// TIA Portal V15.1 export
// export: Created 2024-06-21T08:41:07.2186582Z, ExportSetting WithDefaults, DisplayName Totally Integrated Automation Portal, DisplayVersion V15.1 Update 5, DisplayName TIA Portal Openness, DisplayVersion V15.1 Update 5, DisplayName SINAMICS Startdrive Advanced, DisplayVersion V15.1, DisplayName G130, G150, S120, S150, SINAMICS MV, S210, DisplayVersion V15.1, DisplayName G110M, G120, G120C, G120D, G120P, DisplayVersion V15.1, DisplayName STEP 7 Professional, DisplayVersion V15.1 Update 5, DisplayName STEP 7 Safety, DisplayVersion V15.1, DisplayName WinCC Professional, DisplayVersion V15.1 Update 5, DisplayName SIMATIC Visualization Architect, DisplayVersion V15.1
FUNCTION_BLOCK "LGBHandHeldHBA"   // FB6712, FBD
TITLE = LGBHandHeldHBA
{ S7_Optimized_Access := 'FALSE' }
AUTHOR : VCG
FAMILY : OPanel
VERSION : 1.0
// stored: AutoNumber false, IsIECCheckEnabled false, SetENOAutomatically False, UDAEnableTagReadback false
   VAR_INPUT
      I_HMINbrHandHeld { ExternalAccessible := 'False'; ExternalVisible := 'False'; ExternalWritable := 'False'} : Int;   // HMI number on the function block ModeSelectorHW
      I_ActiveHMI { ExternalAccessible := 'False'; ExternalVisible := 'False'; ExternalWritable := 'False'} : Int;   // Active HMI in the ModeSelectorHW
      I_Connected { ExternalAccessible := 'False'; ExternalVisible := 'False'; ExternalWritable := 'False'} : Bool;   // HandHeld is connected
      I_DeathmansSwitch { ExternalAccessible := 'False'; ExternalVisible := 'False'; ExternalWritable := 'False'} : Bool;   // Deathmans switch
      I_PBSet { ExternalAccessible := 'False'; ExternalVisible := 'False'; ExternalWritable := 'False'} : Bool;   // Push button for manual movememt -> set
      I_PBReset { ExternalAccessible := 'False'; ExternalVisible := 'False'; ExternalWritable := 'False'} : Bool;   // Push button for manual movememt -> reset
      I_PBAlarmReset { ExternalAccessible := 'False'; ExternalVisible := 'False'; ExternalWritable := 'False'} : Bool;   // Push button Alarm reset / Alarm reset pushbutton is activated
      "I_PBSpeed+" { ExternalAccessible := 'False'; ExternalVisible := 'False'; ExternalWritable := 'False'} : Bool;   // Puls for Speed+
      "I_PBSpeed-" { ExternalAccessible := 'False'; ExternalVisible := 'False'; ExternalWritable := 'False'} : Bool;   // Puls for Speed-
      I_PBSelectDevice1 { ExternalAccessible := 'False'; ExternalVisible := 'False'; ExternalWritable := 'False'} : Bool;   // Push button for select Device 1
      I_PBSelectDevice2 { ExternalAccessible := 'False'; ExternalVisible := 'False'; ExternalWritable := 'False'} : Bool;   // Push button for select Device 2
      I_PBSelectDevice3 { ExternalAccessible := 'False'; ExternalVisible := 'False'; ExternalWritable := 'False'} : Bool;   // Push button for select Device 3
      I_PBSelectDevice4 { ExternalAccessible := 'False'; ExternalVisible := 'False'; ExternalWritable := 'False'} : Bool;   // Push button for select Device 4
      I_PBSelectDevice5 { ExternalAccessible := 'False'; ExternalVisible := 'False'; ExternalWritable := 'False'} : Bool;   // Push button for select Device 5
      I_PBSelectDevice6 { ExternalAccessible := 'False'; ExternalVisible := 'False'; ExternalWritable := 'False'} : Bool;   // Push button for select Device 6
      I_PBSelectDevice7 { ExternalAccessible := 'False'; ExternalVisible := 'False'; ExternalWritable := 'False'} : Bool;   // Push button for select Device7
      I_PBSelectDevice8 { ExternalAccessible := 'False'; ExternalVisible := 'False'; ExternalWritable := 'False'} : Bool;   // Push button for select Device 8
      I_PBSelectDevice9 { ExternalAccessible := 'False'; ExternalVisible := 'False'; ExternalWritable := 'False'} : Bool;   // Push button for select Device 9
      I_ActiveDevice1 { ExternalAccessible := 'False'; ExternalVisible := 'False'; ExternalWritable := 'False'} : Bool;   // Device 1 is active
      I_ActiveDevice2 { ExternalAccessible := 'False'; ExternalVisible := 'False'; ExternalWritable := 'False'} : Bool;   // Device 2 is active
      I_ActiveDevice3 { ExternalAccessible := 'False'; ExternalVisible := 'False'; ExternalWritable := 'False'} : Bool;   // Device 3 is active
      I_ActiveDevice4 { ExternalAccessible := 'False'; ExternalVisible := 'False'; ExternalWritable := 'False'} : Bool;   // Device 4 is active
      I_ActiveDevice5 { ExternalAccessible := 'False'; ExternalVisible := 'False'; ExternalWritable := 'False'} : Bool;   // Device 5 is active
      I_ActiveDevice6 { ExternalAccessible := 'False'; ExternalVisible := 'False'; ExternalWritable := 'False'} : Bool;   // Device 6 is active
      I_ActiveDevice7 { ExternalAccessible := 'False'; ExternalVisible := 'False'; ExternalWritable := 'False'} : Bool;   // Device 7 is active
      I_ActiveDevice8 { ExternalAccessible := 'False'; ExternalVisible := 'False'; ExternalWritable := 'False'} : Bool;   // Device 8 is active
      I_ActiveDevice9 { ExternalAccessible := 'False'; ExternalVisible := 'False'; ExternalWritable := 'False'} : Bool;   // Device 9 is active
      I_LEDAlarmReset { ExternalAccessible := 'False'; ExternalVisible := 'False'; ExternalWritable := 'False'} : Bool;   // Led Indication Push button Alarm reset / Alarm reset pushbutton is activated
   END_VAR
   VAR_OUTPUT
      O_HandHeldConnected { ExternalAccessible := 'False'; ExternalVisible := 'False'; ExternalWritable := 'False'} : Bool;   // HandHeld is connected
      O_HandHeldSelected { ExternalAccessible := 'False'; ExternalVisible := 'False'; ExternalWritable := 'False'} : Bool;   // HandHeld is selected, is active HMI
      O_AlarmReset { ExternalAccessible := 'False'; ExternalVisible := 'False'; ExternalWritable := 'False'} : Bool;   // Push button Alarm reset / Alarm reset pushbutton is activated
      O_Speed { ExternalAccessible := 'False'; ExternalVisible := 'False'; ExternalWritable := 'False'} : Int;   // Speed
      "O_Speed+" { ExternalAccessible := 'False'; ExternalVisible := 'False'; ExternalWritable := 'False'} : Bool;   // Push button Speed+
      "O_Speed-" { ExternalAccessible := 'False'; ExternalVisible := 'False'; ExternalWritable := 'False'} : Bool;   // Push button Speed-
      O_HighSpeed { ExternalAccessible := 'False'; ExternalVisible := 'False'; ExternalWritable := 'False'} : Bool;   // High Speed Selected
      O_PBSetDevice1 { ExternalAccessible := 'False'; ExternalVisible := 'False'; ExternalWritable := 'False'} : Bool;   // Device 1 Push button Set
      O_PBResDevice1 { ExternalAccessible := 'False'; ExternalVisible := 'False'; ExternalWritable := 'False'} : Bool;   // Device 1 Push button Reset
      O_PBSetDevice2 { ExternalAccessible := 'False'; ExternalVisible := 'False'; ExternalWritable := 'False'} : Bool;   // Device 2 Push button Set
      O_PBResDevice2 { ExternalAccessible := 'False'; ExternalVisible := 'False'; ExternalWritable := 'False'} : Bool;   // Device 2 Push button Reset
      O_PBSetDevice3 { ExternalAccessible := 'False'; ExternalVisible := 'False'; ExternalWritable := 'False'} : Bool;   // Device 3 Push button Set
      O_PBResDevice3 { ExternalAccessible := 'False'; ExternalVisible := 'False'; ExternalWritable := 'False'} : Bool;   // Device 3 Push button Reset
      O_PBSetDevice4 { ExternalAccessible := 'False'; ExternalVisible := 'False'; ExternalWritable := 'False'} : Bool;   // Device 4 Push button Set
      O_PBResDevice4 { ExternalAccessible := 'False'; ExternalVisible := 'False'; ExternalWritable := 'False'} : Bool;   // Device 4 Push button Reset
      O_PBSetDevice5 { ExternalAccessible := 'False'; ExternalVisible := 'False'; ExternalWritable := 'False'} : Bool;   // Device 5 Push button Set
      O_PBResDevice5 { ExternalAccessible := 'False'; ExternalVisible := 'False'; ExternalWritable := 'False'} : Bool;   // Device 5 Push button Reset
      O_PBSetDevice6 { ExternalAccessible := 'False'; ExternalVisible := 'False'; ExternalWritable := 'False'} : Bool;   // Device 6 Push button Set
      O_PBResDevice6 { ExternalAccessible := 'False'; ExternalVisible := 'False'; ExternalWritable := 'False'} : Bool;   // Device 6 Push button Reset
      O_PBSetDevice7 { ExternalAccessible := 'False'; ExternalVisible := 'False'; ExternalWritable := 'False'} : Bool;   // Device 7 Push button Set
      O_PBResDevice7 { ExternalAccessible := 'False'; ExternalVisible := 'False'; ExternalWritable := 'False'} : Bool;   // Device 7 Push button Reset
      O_PBSetDevice8 { ExternalAccessible := 'False'; ExternalVisible := 'False'; ExternalWritable := 'False'} : Bool;   // Device 8 Push button Set
      O_PBResDevice8 { ExternalAccessible := 'False'; ExternalVisible := 'False'; ExternalWritable := 'False'} : Bool;   // Device 8 Push button Reset
      O_PBSetDevice9 { ExternalAccessible := 'False'; ExternalVisible := 'False'; ExternalWritable := 'False'} : Bool;   // Device 9 Push button Set
      O_PBResDevice9 { ExternalAccessible := 'False'; ExternalVisible := 'False'; ExternalWritable := 'False'} : Bool;   // Device 9 Push button Reset
      O_LEDSet { ExternalAccessible := 'False'; ExternalVisible := 'False'; ExternalWritable := 'False'} : Bool;   // Led Indication Push button set
      O_LEDReset { ExternalAccessible := 'False'; ExternalVisible := 'False'; ExternalWritable := 'False'} : Bool;   // Led Indication Push button reset
      O_LEDAlarmReset { ExternalAccessible := 'False'; ExternalVisible := 'False'; ExternalWritable := 'False'} : Bool;   // Led Indication Push button Alarm reset / Alarm reset pushbutton is activated
      "O_LEDSpeed+" { ExternalAccessible := 'False'; ExternalVisible := 'False'; ExternalWritable := 'False'} : Bool;   // Led Indication Puls Speed+
      "O_LEDSpeed-" { ExternalAccessible := 'False'; ExternalVisible := 'False'; ExternalWritable := 'False'} : Bool;   // Led Indication Puls Speed-
      O_LEDDevice1 { ExternalAccessible := 'False'; ExternalVisible := 'False'; ExternalWritable := 'False'} : Bool;   // Led Indication Push button Device 1
      O_LEDDevice2 { ExternalAccessible := 'False'; ExternalVisible := 'False'; ExternalWritable := 'False'} : Bool;   // Led Indication Push button Device 2
      O_LEDDevice3 { ExternalAccessible := 'False'; ExternalVisible := 'False'; ExternalWritable := 'False'} : Bool;   // Led Indication Push button Device 3
      O_LEDDevice4 { ExternalAccessible := 'False'; ExternalVisible := 'False'; ExternalWritable := 'False'} : Bool;   // Led Indication Push button Device 4
      O_LEDDevice5 { ExternalAccessible := 'False'; ExternalVisible := 'False'; ExternalWritable := 'False'} : Bool;   // Led Indication Push button Device 5
      O_LEDDevice6 { ExternalAccessible := 'False'; ExternalVisible := 'False'; ExternalWritable := 'False'} : Bool;   // Led Indication Push button Device 6
      O_LEDDevice7 { ExternalAccessible := 'False'; ExternalVisible := 'False'; ExternalWritable := 'False'} : Bool;   // Led Indication Push button Device 7
      O_LEDDevice8 { ExternalAccessible := 'False'; ExternalVisible := 'False'; ExternalWritable := 'False'} : Bool;   // Led Indication Push button Device 8
      O_LEDDevice9 { ExternalAccessible := 'False'; ExternalVisible := 'False'; ExternalWritable := 'False'} : Bool;   // Led Indication Push button Device 9
   END_VAR
   VAR_IN_OUT
      IO_Modes : "Modes";   // Modes IO
      C_Config : "HandHeldHBA-Config";   // Config
   END_VAR
   VAR DB_SPECIFIC
      HandHeldSelected { ExternalAccessible := 'False'; ExternalVisible := 'False'; ExternalWritable := 'False'} : Bool;   // HandHeld is selected, is active HMI
      HighSpeed { ExternalAccessible := 'False'; ExternalVisible := 'False'; ExternalWritable := 'False'} : Bool;   // High Speed Selected
      Device1SelectedForHighSpeed { ExternalAccessible := 'False'; ExternalVisible := 'False'; ExternalWritable := 'False'} : Bool;   // Device 1 is selected for High speed
      Device2SelectedForHighSpeed { ExternalAccessible := 'False'; ExternalVisible := 'False'; ExternalWritable := 'False'} : Bool;   // Device 2 is selected for High speed
      Device3SelectedForHighSpeed { ExternalAccessible := 'False'; ExternalVisible := 'False'; ExternalWritable := 'False'} : Bool;   // Device 3 is selected for High speed
      Device4SelectedForHighSpeed { ExternalAccessible := 'False'; ExternalVisible := 'False'; ExternalWritable := 'False'} : Bool;   // Device 4 is selected for High speed
      Device5SelectedForHighSpeed { ExternalAccessible := 'False'; ExternalVisible := 'False'; ExternalWritable := 'False'} : Bool;   // Device 5 is selected for High speed
      Device6SelectedForHighSpeed { ExternalAccessible := 'False'; ExternalVisible := 'False'; ExternalWritable := 'False'} : Bool;   // Device 6 is selected for High speed
      Device7SelectedForHighSpeed { ExternalAccessible := 'False'; ExternalVisible := 'False'; ExternalWritable := 'False'} : Bool;   // Device 7 is selected for High speed
      Device8SelectedForHighSpeed { ExternalAccessible := 'False'; ExternalVisible := 'False'; ExternalWritable := 'False'} : Bool;   // Device 8 is selected for High speed
      Device9SelectedForHighSpeed { ExternalAccessible := 'False'; ExternalVisible := 'False'; ExternalWritable := 'False'} : Bool;   // Device 9 is selected for High speed
      Device1Selected { ExternalAccessible := 'False'; ExternalVisible := 'False'; ExternalWritable := 'False'} : Bool;   // Device 1 is selected
      Device2Selected { ExternalAccessible := 'False'; ExternalVisible := 'False'; ExternalWritable := 'False'} : Bool;   // Device 2 is selected
      Device3Selected { ExternalAccessible := 'False'; ExternalVisible := 'False'; ExternalWritable := 'False'} : Bool;   // Device 3 is selected
      Device4Selected { ExternalAccessible := 'False'; ExternalVisible := 'False'; ExternalWritable := 'False'} : Bool;   // Device 4 is selected
      Device5Selected { ExternalAccessible := 'False'; ExternalVisible := 'False'; ExternalWritable := 'False'} : Bool;   // Device 5 is selected
      Device6Selected { ExternalAccessible := 'False'; ExternalVisible := 'False'; ExternalWritable := 'False'} : Bool;   // Device 6 is selected
      Device7Selected { ExternalAccessible := 'False'; ExternalVisible := 'False'; ExternalWritable := 'False'} : Bool;   // Device 7 is selected
      Device8Selected { ExternalAccessible := 'False'; ExternalVisible := 'False'; ExternalWritable := 'False'} : Bool;   // Device 8 is selected
      Device9Selected { ExternalAccessible := 'False'; ExternalVisible := 'False'; ExternalWritable := 'False'} : Bool;   // Device 9 is selected
      PBSetDevice1 { ExternalAccessible := 'False'; ExternalVisible := 'False'; ExternalWritable := 'False'} : Bool;   // Device 1 Push button Set
      PBResDevice1 { ExternalAccessible := 'False'; ExternalVisible := 'False'; ExternalWritable := 'False'} : Bool;   // Device 1 Push button Reset
      PBSetDevice2 { ExternalAccessible := 'False'; ExternalVisible := 'False'; ExternalWritable := 'False'} : Bool;   // Device 2 Push button Set
      PBResDevice2 { ExternalAccessible := 'False'; ExternalVisible := 'False'; ExternalWritable := 'False'} : Bool;   // Device 2 Push button Reset
      PBSetDevice3 { ExternalAccessible := 'False'; ExternalVisible := 'False'; ExternalWritable := 'False'} : Bool;   // Device 3 Push button Set
      PBResDevice3 { ExternalAccessible := 'False'; ExternalVisible := 'False'; ExternalWritable := 'False'} : Bool;   // Device 3 Push button Reset
      PBSetDevice4 { ExternalAccessible := 'False'; ExternalVisible := 'False'; ExternalWritable := 'False'} : Bool;   // Device 4 Push button Set
      PBResDevice4 { ExternalAccessible := 'False'; ExternalVisible := 'False'; ExternalWritable := 'False'} : Bool;   // Device 4 Push button Reset
      PBSetDevice5 { ExternalAccessible := 'False'; ExternalVisible := 'False'; ExternalWritable := 'False'} : Bool;   // Device 5 Push button Set
      PBResDevice5 { ExternalAccessible := 'False'; ExternalVisible := 'False'; ExternalWritable := 'False'} : Bool;   // Device 5 Push button Reset
      PBSetDevice6 { ExternalAccessible := 'False'; ExternalVisible := 'False'; ExternalWritable := 'False'} : Bool;   // Device 6 Push button Set
      PBResDevice6 { ExternalAccessible := 'False'; ExternalVisible := 'False'; ExternalWritable := 'False'} : Bool;   // Device 6 Push button Reset
      PBSetDevice7 { ExternalAccessible := 'False'; ExternalVisible := 'False'; ExternalWritable := 'False'} : Bool;   // Device 7 Push button Set
      PBResDevice7 { ExternalAccessible := 'False'; ExternalVisible := 'False'; ExternalWritable := 'False'} : Bool;   // Device 7 Push button Reset
      PBSetDevice8 { ExternalAccessible := 'False'; ExternalVisible := 'False'; ExternalWritable := 'False'} : Bool;   // Device 8 Push button Set
      PBResDevice8 { ExternalAccessible := 'False'; ExternalVisible := 'False'; ExternalWritable := 'False'} : Bool;   // Device 8 Push button Reset
      PBSetDevice9 { ExternalAccessible := 'False'; ExternalVisible := 'False'; ExternalWritable := 'False'} : Bool;   // Device 9 Push button Set
      PBResDevice9 { ExternalAccessible := 'False'; ExternalVisible := 'False'; ExternalWritable := 'False'} : Bool;   // Device 9 Push button Reset
      LEDDevice1 { ExternalAccessible := 'False'; ExternalVisible := 'False'; ExternalWritable := 'False'} : Bool;   // Indication Push button Device 1
      LEDDevice2 { ExternalAccessible := 'False'; ExternalVisible := 'False'; ExternalWritable := 'False'} : Bool;   // Indication Push button Device 2
      LEDDevice3 { ExternalAccessible := 'False'; ExternalVisible := 'False'; ExternalWritable := 'False'} : Bool;   // Indication Push button Device 3
      LEDDevice4 { ExternalAccessible := 'False'; ExternalVisible := 'False'; ExternalWritable := 'False'} : Bool;   // Indication Push button Device 4
      LEDDevice5 { ExternalAccessible := 'False'; ExternalVisible := 'False'; ExternalWritable := 'False'} : Bool;   // Indication Push button Device 5
      LEDDevice6 { ExternalAccessible := 'False'; ExternalVisible := 'False'; ExternalWritable := 'False'} : Bool;   // Indication Push button Device 6
      LEDDevice7 { ExternalAccessible := 'False'; ExternalVisible := 'False'; ExternalWritable := 'False'} : Bool;   // Indication Push button Device 7
      LEDDevice8 { ExternalAccessible := 'False'; ExternalVisible := 'False'; ExternalWritable := 'False'} : Bool;   // Indication Push button Device 8
      LEDDevice9 { ExternalAccessible := 'False'; ExternalVisible := 'False'; ExternalWritable := 'False'} : Bool;   // Indication Push button Device 9
      Speed { ExternalAccessible := 'False'; ExternalVisible := 'False'; ExternalWritable := 'False'} : Int;   // Speed
      Edge { ExternalAccessible := 'False'; ExternalVisible := 'False'; ExternalWritable := 'False'} : Array[1..20] of Bool;   // Edge
   END_VAR
   VAR
      Toggle_Device1SelectedForHighSpeed { ExternalAccessible := 'False'; ExternalVisible := 'False'; ExternalWritable := 'False'} : "LToggle";   // FB
      Toggle_Device2SelectedForHighSpeed { ExternalAccessible := 'False'; ExternalVisible := 'False'; ExternalWritable := 'False'} : "LToggle";   // FB
      Toggle_Device3SelectedForHighSpeed { ExternalAccessible := 'False'; ExternalVisible := 'False'; ExternalWritable := 'False'} : "LToggle";   // FB
      Toggle_Device4SelectedForHighSpeed { ExternalAccessible := 'False'; ExternalVisible := 'False'; ExternalWritable := 'False'} : "LToggle";   // FB
      Toggle_Device5SelectedForHighSpeed { ExternalAccessible := 'False'; ExternalVisible := 'False'; ExternalWritable := 'False'} : "LToggle";   // FB
      Toggle_Device6SelectedForHighSpeed { ExternalAccessible := 'False'; ExternalVisible := 'False'; ExternalWritable := 'False'} : "LToggle";   // FB
      Toggle_Device7SelectedForHighSpeed { ExternalAccessible := 'False'; ExternalVisible := 'False'; ExternalWritable := 'False'} : "LToggle";   // FB
      Toggle_Device8SelectedForHighSpeed { ExternalAccessible := 'False'; ExternalVisible := 'False'; ExternalWritable := 'False'} : "LToggle";   // FB
      Toggle_Device9SelectedForHighSpeed { ExternalAccessible := 'False'; ExternalVisible := 'False'; ExternalWritable := 'False'} : "LToggle";   // FB
   END_VAR
   VAR_TEMP   // added for the SCL form of the ladder/FBD networks
      _w1 : Bool;
   END_VAR
BEGIN

REGION Network 1: **** 1 - Inputs **** HandHeld is selected, is active HMI
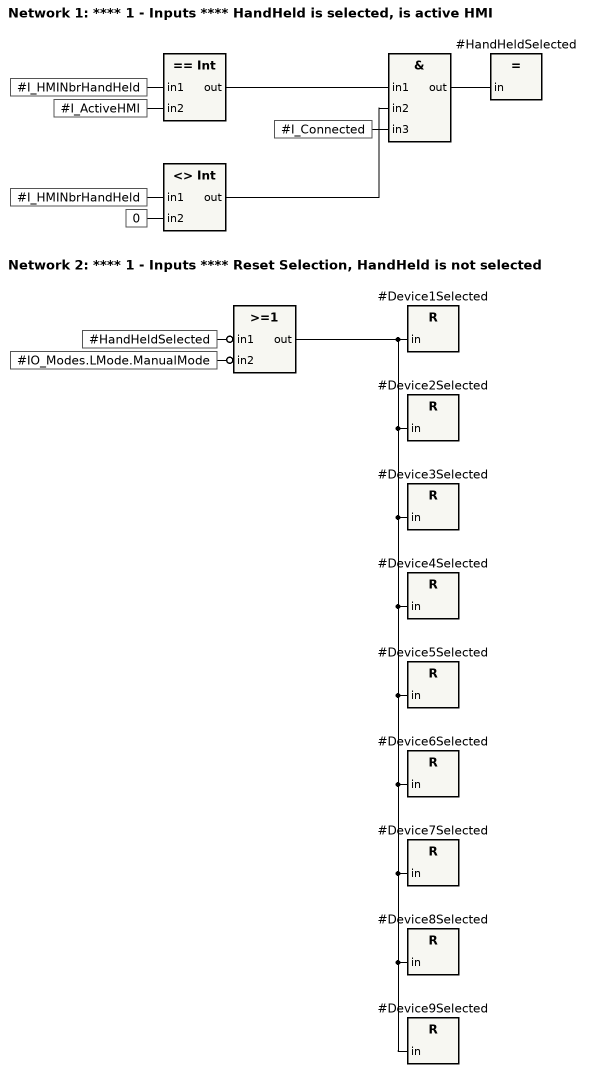
   #HandHeldSelected := (#I_HMINbrHandHeld = #I_ActiveHMI) AND (#I_HMINbrHandHeld <> 0) AND #I_Connected;
END_REGION

REGION Network 2: **** 1 - Inputs **** Reset Selection, HandHeld is not selected
   IF NOT #HandHeldSelected OR NOT #IO_Modes.LMode.ManualMode THEN
       #Device1Selected := FALSE;
       #Device2Selected := FALSE;
       #Device3Selected := FALSE;
       #Device4Selected := FALSE;
       #Device5Selected := FALSE;
       #Device6Selected := FALSE;
       #Device7Selected := FALSE;
       #Device8Selected := FALSE;
       #Device9Selected := FALSE;
   END_IF;
END_REGION

REGION Network 3: **** 4.3 - Machine status - Operator Selection **** Device 1 is selected for High speed
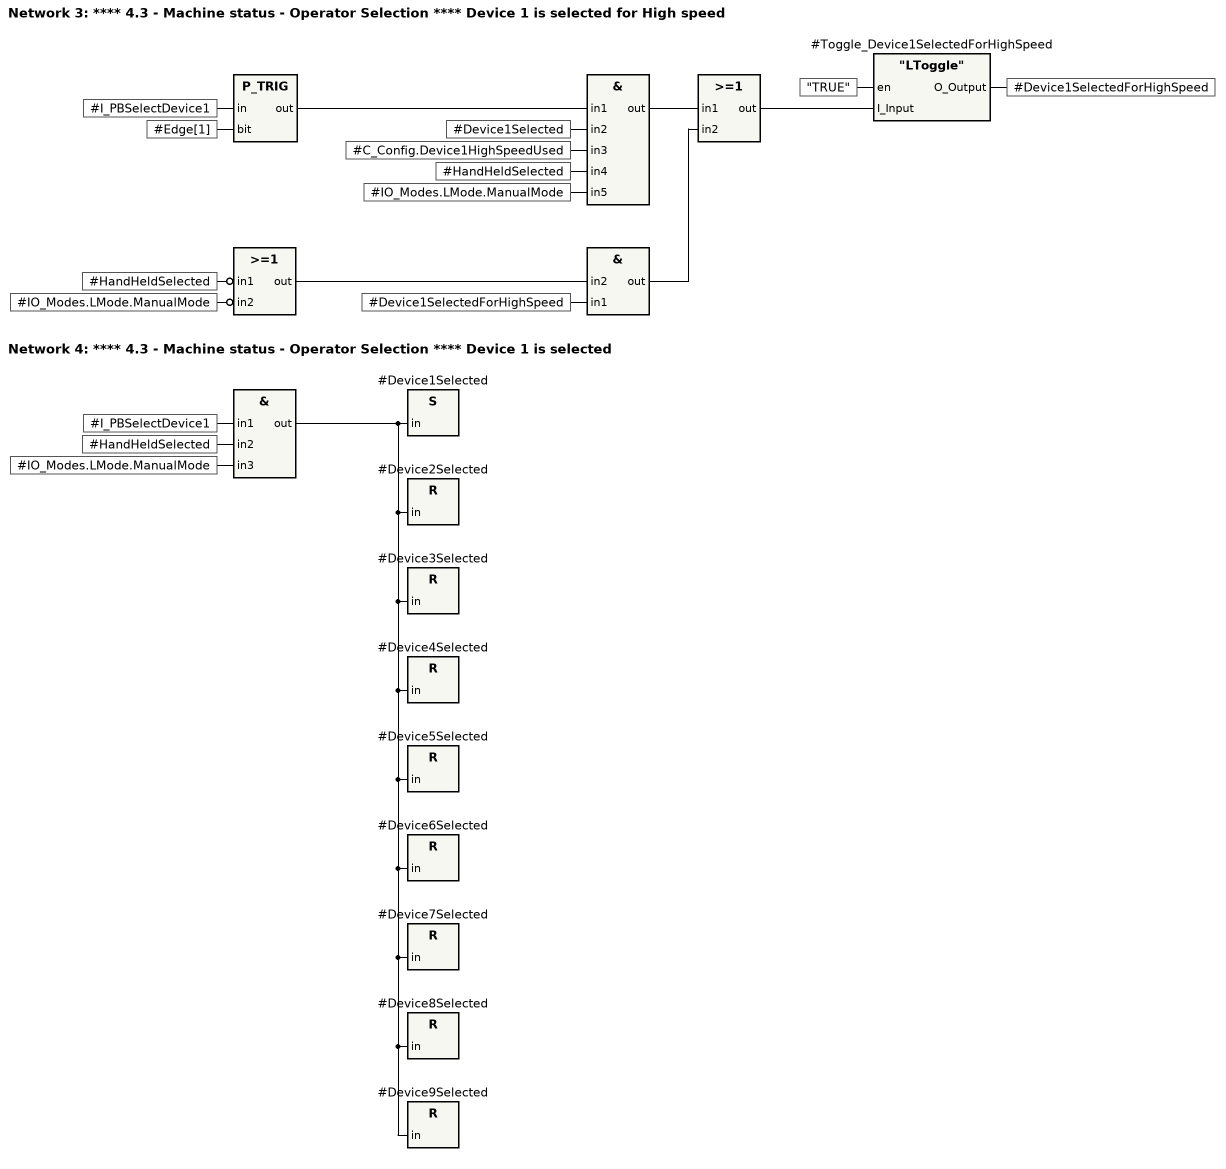
   #_w1 := #I_PBSelectDevice1 AND NOT #Edge[1];   // rising edge
   #Edge[1] := #I_PBSelectDevice1;
   IF "TRUE" THEN
       #Toggle_Device1SelectedForHighSpeed(I_Input := (#_w1 AND #Device1Selected AND #C_Config.Device1HighSpeedUsed AND #HandHeldSelected AND #IO_Modes.LMode.ManualMode) OR ((NOT #HandHeldSelected OR NOT #IO_Modes.LMode.ManualMode) AND #Device1SelectedForHighSpeed),   // "LToggle"
                               O_Output => #Device1SelectedForHighSpeed);
   END_IF;
END_REGION

REGION Network 4: **** 4.3 - Machine status - Operator Selection **** Device 1 is selected
   IF #I_PBSelectDevice1 AND #HandHeldSelected AND #IO_Modes.LMode.ManualMode THEN
       #Device1Selected := TRUE;
       #Device2Selected := FALSE;
       #Device3Selected := FALSE;
       #Device4Selected := FALSE;
       #Device5Selected := FALSE;
       #Device6Selected := FALSE;
       #Device7Selected := FALSE;
       #Device8Selected := FALSE;
       #Device9Selected := FALSE;
   END_IF;
END_REGION

REGION Network 5: **** 4.3 - Machine status - Operator Selection **** Device 2 is selected for High speed
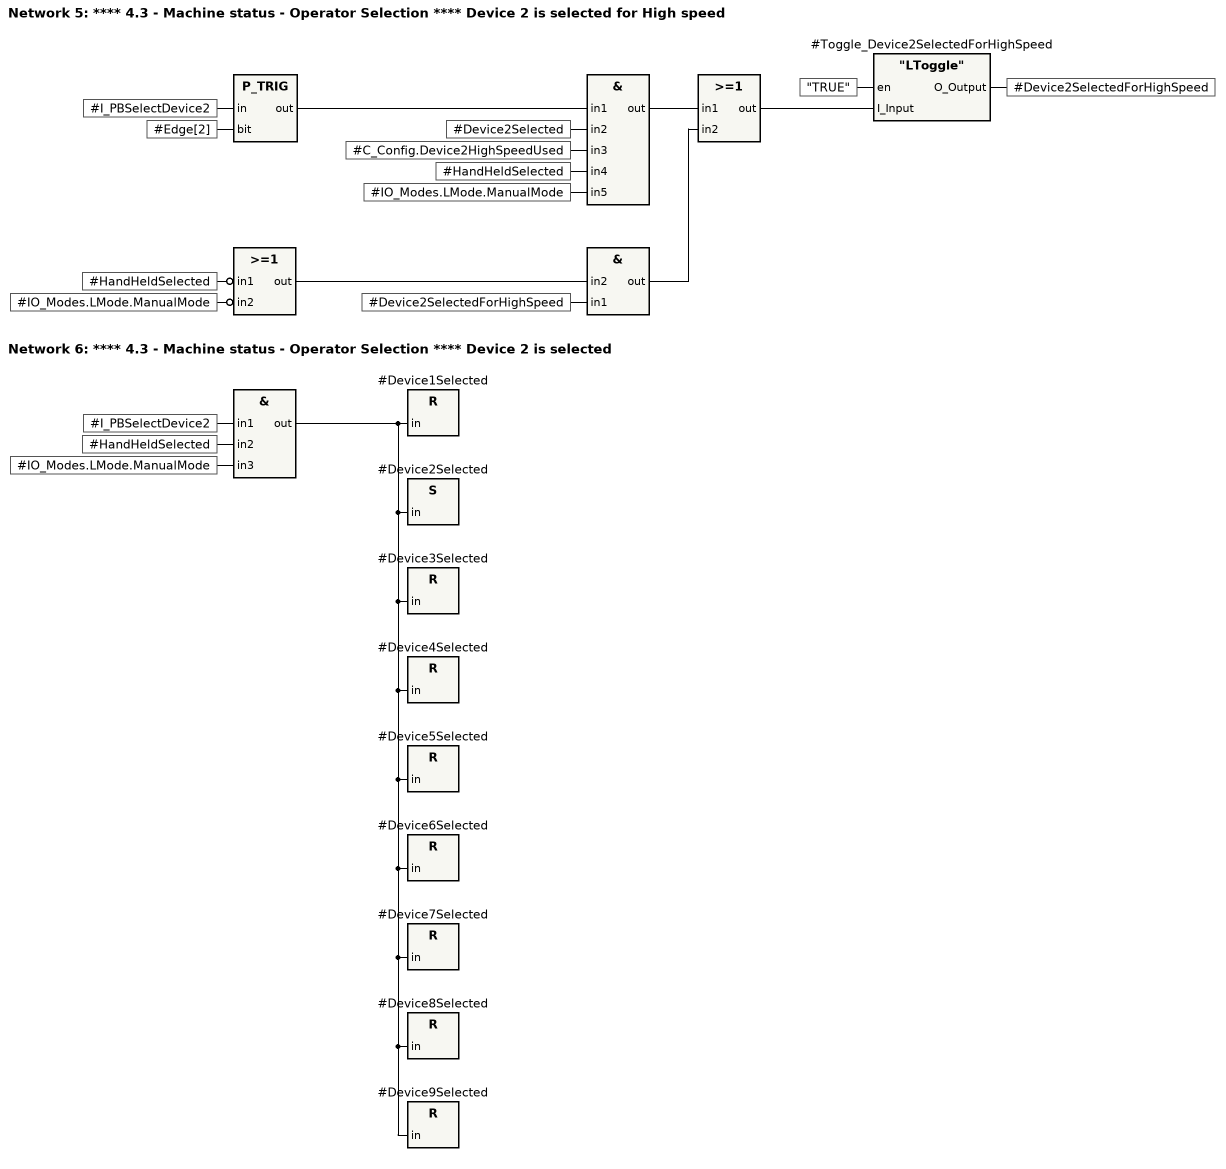
   #_w1 := #I_PBSelectDevice2 AND NOT #Edge[2];   // rising edge
   #Edge[2] := #I_PBSelectDevice2;
   IF "TRUE" THEN
       #Toggle_Device2SelectedForHighSpeed(I_Input := (#_w1 AND #Device2Selected AND #C_Config.Device2HighSpeedUsed AND #HandHeldSelected AND #IO_Modes.LMode.ManualMode) OR ((NOT #HandHeldSelected OR NOT #IO_Modes.LMode.ManualMode) AND #Device2SelectedForHighSpeed),   // "LToggle"
                               O_Output => #Device2SelectedForHighSpeed);
   END_IF;
END_REGION

REGION Network 6: **** 4.3 - Machine status - Operator Selection **** Device 2 is selected
   IF #I_PBSelectDevice2 AND #HandHeldSelected AND #IO_Modes.LMode.ManualMode THEN
       #Device1Selected := FALSE;
       #Device2Selected := TRUE;
       #Device3Selected := FALSE;
       #Device4Selected := FALSE;
       #Device5Selected := FALSE;
       #Device6Selected := FALSE;
       #Device7Selected := FALSE;
       #Device8Selected := FALSE;
       #Device9Selected := FALSE;
   END_IF;
END_REGION

REGION Network 7: **** 4.3 - Machine status - Operator Selection **** Device 3 is selected for High speed
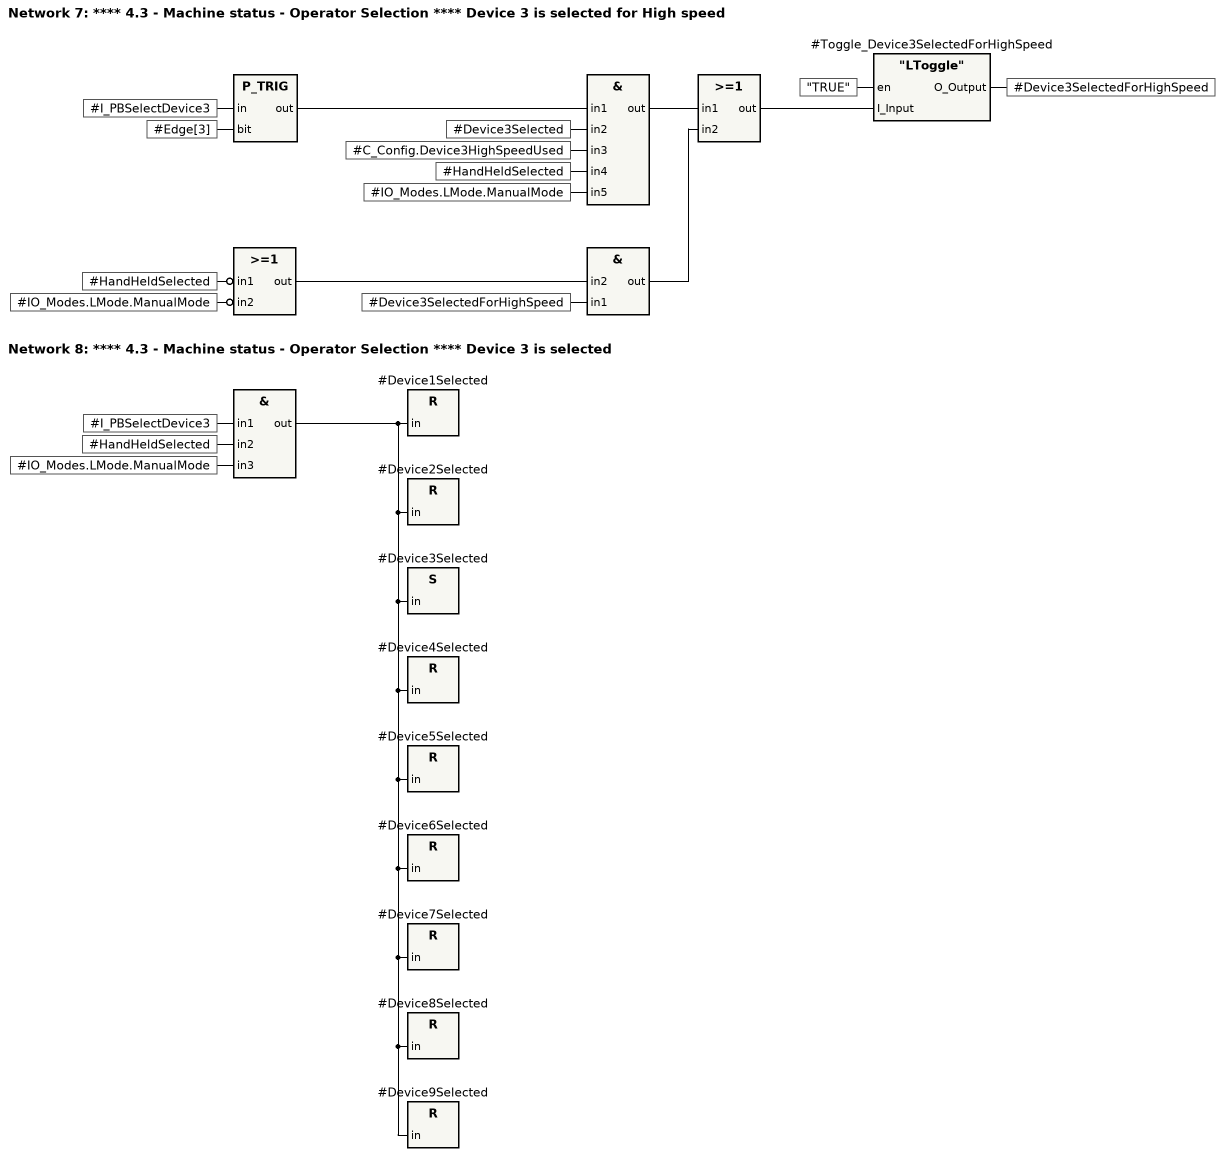
   #_w1 := #I_PBSelectDevice3 AND NOT #Edge[3];   // rising edge
   #Edge[3] := #I_PBSelectDevice3;
   IF "TRUE" THEN
       #Toggle_Device3SelectedForHighSpeed(I_Input := (#_w1 AND #Device3Selected AND #C_Config.Device3HighSpeedUsed AND #HandHeldSelected AND #IO_Modes.LMode.ManualMode) OR ((NOT #HandHeldSelected OR NOT #IO_Modes.LMode.ManualMode) AND #Device3SelectedForHighSpeed),   // "LToggle"
                               O_Output => #Device3SelectedForHighSpeed);
   END_IF;
END_REGION

REGION Network 8: **** 4.3 - Machine status - Operator Selection **** Device 3 is selected
   IF #I_PBSelectDevice3 AND #HandHeldSelected AND #IO_Modes.LMode.ManualMode THEN
       #Device1Selected := FALSE;
       #Device2Selected := FALSE;
       #Device3Selected := TRUE;
       #Device4Selected := FALSE;
       #Device5Selected := FALSE;
       #Device6Selected := FALSE;
       #Device7Selected := FALSE;
       #Device8Selected := FALSE;
       #Device9Selected := FALSE;
   END_IF;
END_REGION

REGION Network 9: **** 4.3 - Machine status - Operator Selection **** Device 4 is selected for High speed
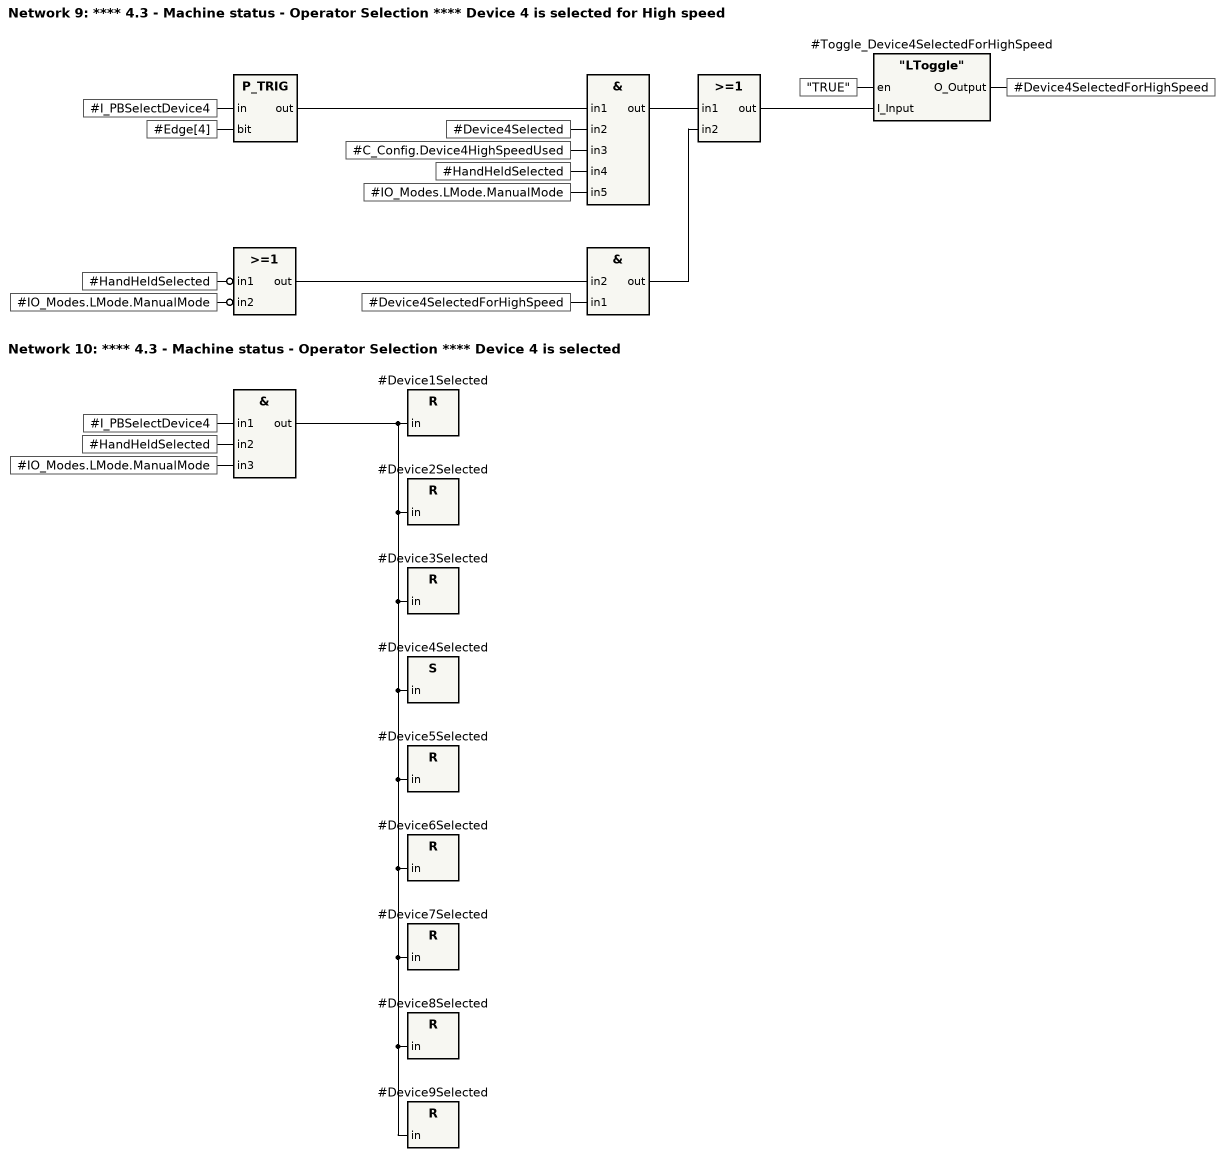
   #_w1 := #I_PBSelectDevice4 AND NOT #Edge[4];   // rising edge
   #Edge[4] := #I_PBSelectDevice4;
   IF "TRUE" THEN
       #Toggle_Device4SelectedForHighSpeed(I_Input := (#_w1 AND #Device4Selected AND #C_Config.Device4HighSpeedUsed AND #HandHeldSelected AND #IO_Modes.LMode.ManualMode) OR ((NOT #HandHeldSelected OR NOT #IO_Modes.LMode.ManualMode) AND #Device4SelectedForHighSpeed),   // "LToggle"
                               O_Output => #Device4SelectedForHighSpeed);
   END_IF;
END_REGION

REGION Network 10: **** 4.3 - Machine status - Operator Selection **** Device 4 is selected
   IF #I_PBSelectDevice4 AND #HandHeldSelected AND #IO_Modes.LMode.ManualMode THEN
       #Device1Selected := FALSE;
       #Device2Selected := FALSE;
       #Device3Selected := FALSE;
       #Device4Selected := TRUE;
       #Device5Selected := FALSE;
       #Device6Selected := FALSE;
       #Device7Selected := FALSE;
       #Device8Selected := FALSE;
       #Device9Selected := FALSE;
   END_IF;
END_REGION

REGION Network 11: **** 4.3 - Machine status - Operator Selection **** Device 5 is selected for High speed
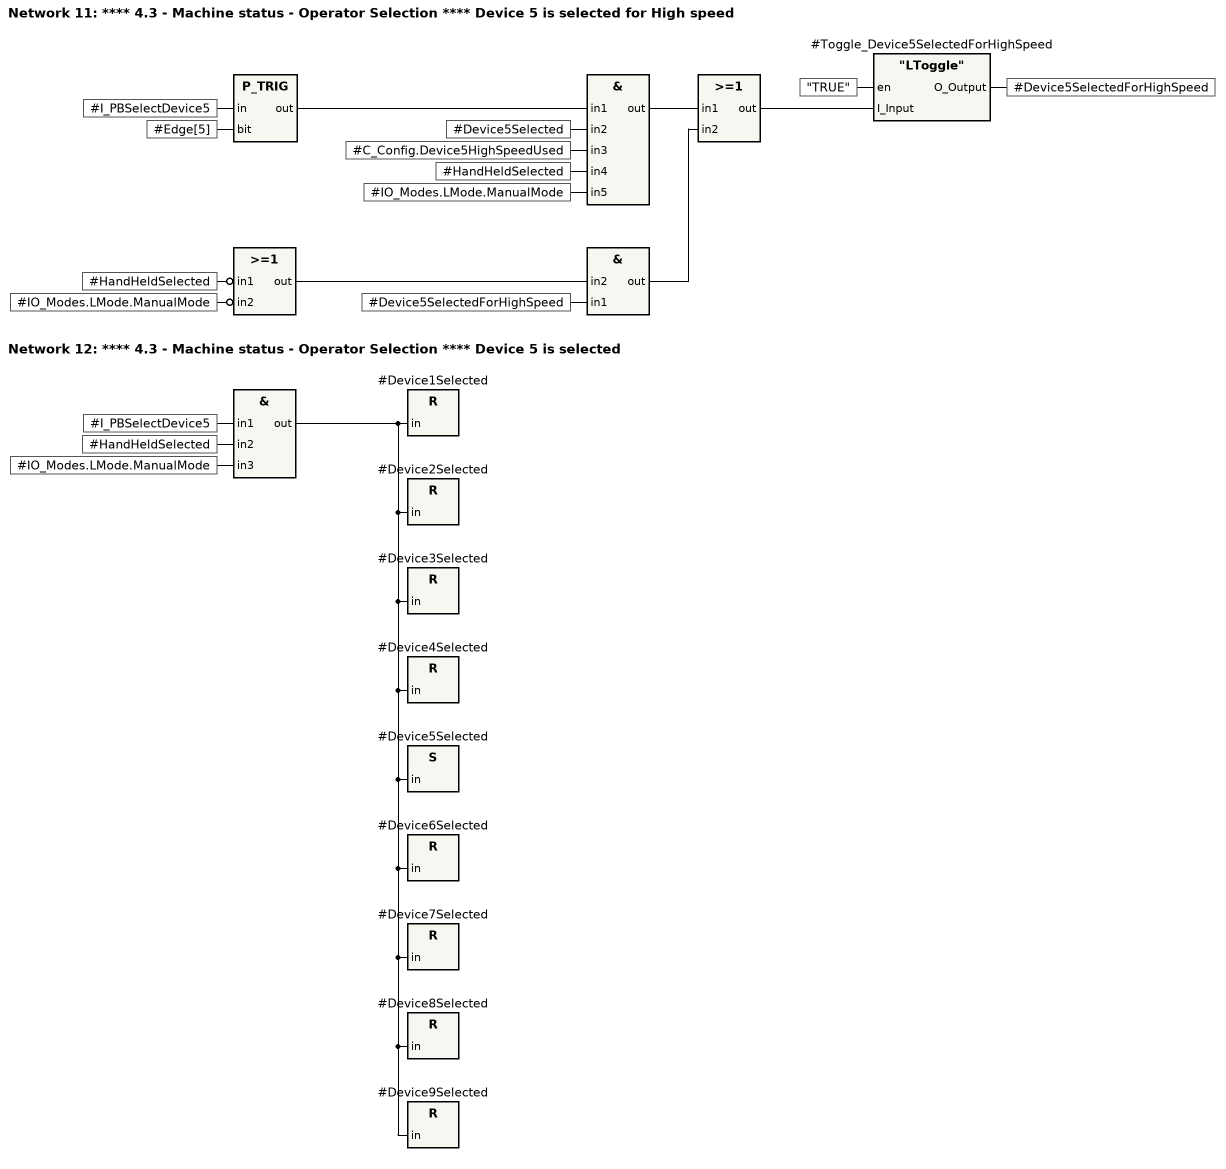
   #_w1 := #I_PBSelectDevice5 AND NOT #Edge[5];   // rising edge
   #Edge[5] := #I_PBSelectDevice5;
   IF "TRUE" THEN
       #Toggle_Device5SelectedForHighSpeed(I_Input := (#_w1 AND #Device5Selected AND #C_Config.Device5HighSpeedUsed AND #HandHeldSelected AND #IO_Modes.LMode.ManualMode) OR ((NOT #HandHeldSelected OR NOT #IO_Modes.LMode.ManualMode) AND #Device5SelectedForHighSpeed),   // "LToggle"
                               O_Output => #Device5SelectedForHighSpeed);
   END_IF;
END_REGION

REGION Network 12: **** 4.3 - Machine status - Operator Selection **** Device 5 is selected
   IF #I_PBSelectDevice5 AND #HandHeldSelected AND #IO_Modes.LMode.ManualMode THEN
       #Device1Selected := FALSE;
       #Device2Selected := FALSE;
       #Device3Selected := FALSE;
       #Device4Selected := FALSE;
       #Device5Selected := TRUE;
       #Device6Selected := FALSE;
       #Device7Selected := FALSE;
       #Device8Selected := FALSE;
       #Device9Selected := FALSE;
   END_IF;
END_REGION

REGION Network 13: **** 4.3 - Machine status - Operator Selection **** Device 6 is selected for High speed
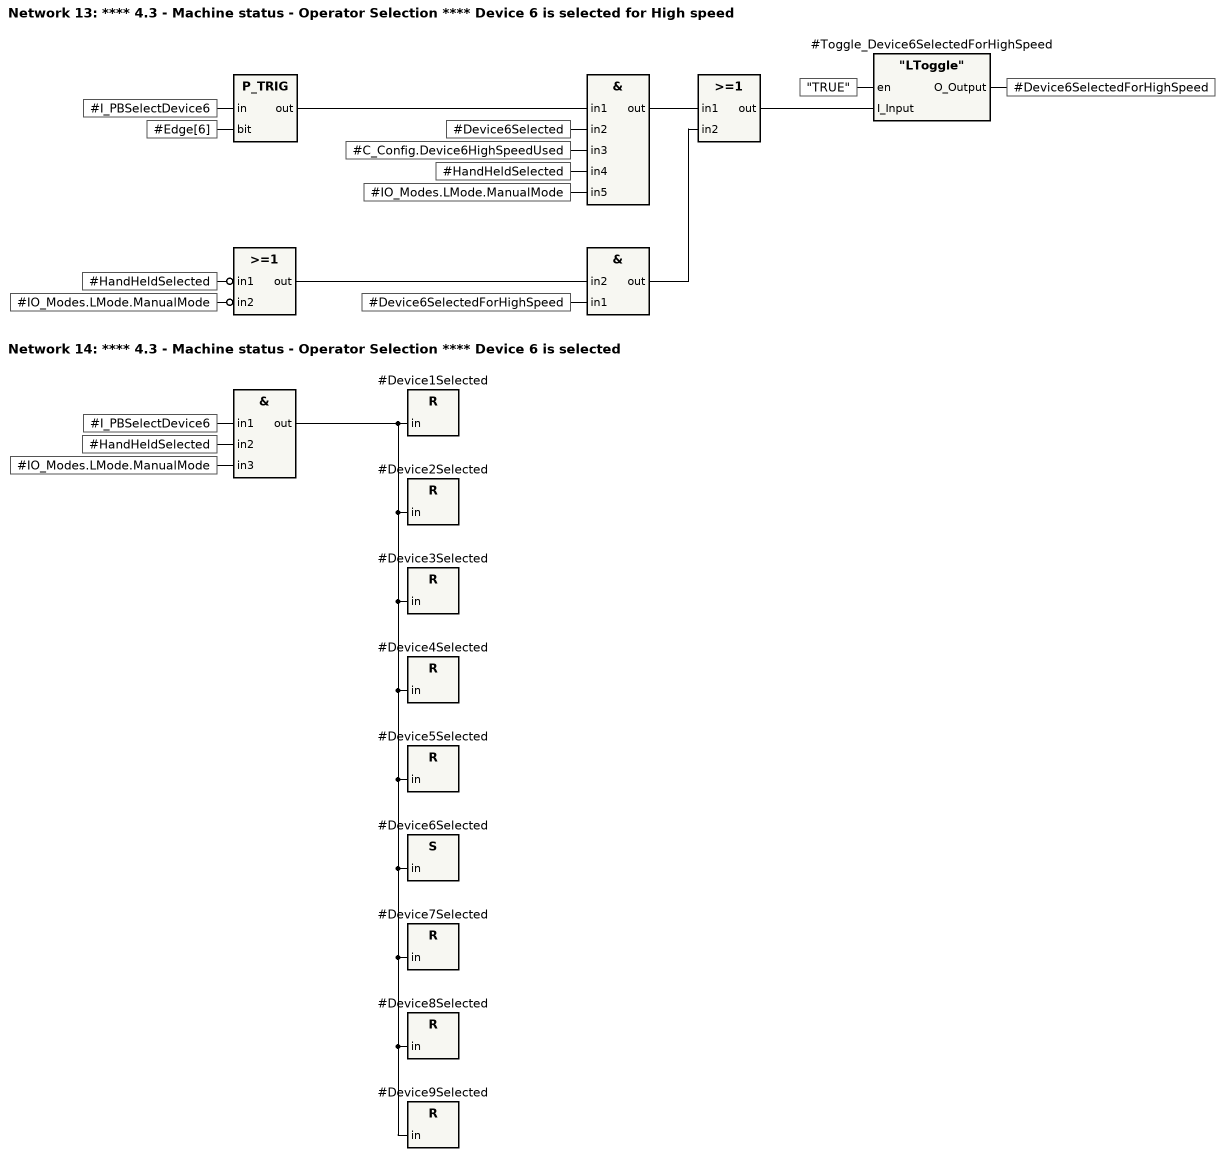
   #_w1 := #I_PBSelectDevice6 AND NOT #Edge[6];   // rising edge
   #Edge[6] := #I_PBSelectDevice6;
   IF "TRUE" THEN
       #Toggle_Device6SelectedForHighSpeed(I_Input := (#_w1 AND #Device6Selected AND #C_Config.Device6HighSpeedUsed AND #HandHeldSelected AND #IO_Modes.LMode.ManualMode) OR ((NOT #HandHeldSelected OR NOT #IO_Modes.LMode.ManualMode) AND #Device6SelectedForHighSpeed),   // "LToggle"
                               O_Output => #Device6SelectedForHighSpeed);
   END_IF;
END_REGION

REGION Network 14: **** 4.3 - Machine status - Operator Selection **** Device 6 is selected
   IF #I_PBSelectDevice6 AND #HandHeldSelected AND #IO_Modes.LMode.ManualMode THEN
       #Device1Selected := FALSE;
       #Device2Selected := FALSE;
       #Device3Selected := FALSE;
       #Device4Selected := FALSE;
       #Device5Selected := FALSE;
       #Device6Selected := TRUE;
       #Device7Selected := FALSE;
       #Device8Selected := FALSE;
       #Device9Selected := FALSE;
   END_IF;
END_REGION

REGION Network 15: **** 4.3 - Machine status - Operator Selection **** Device 7 is selected for High speed
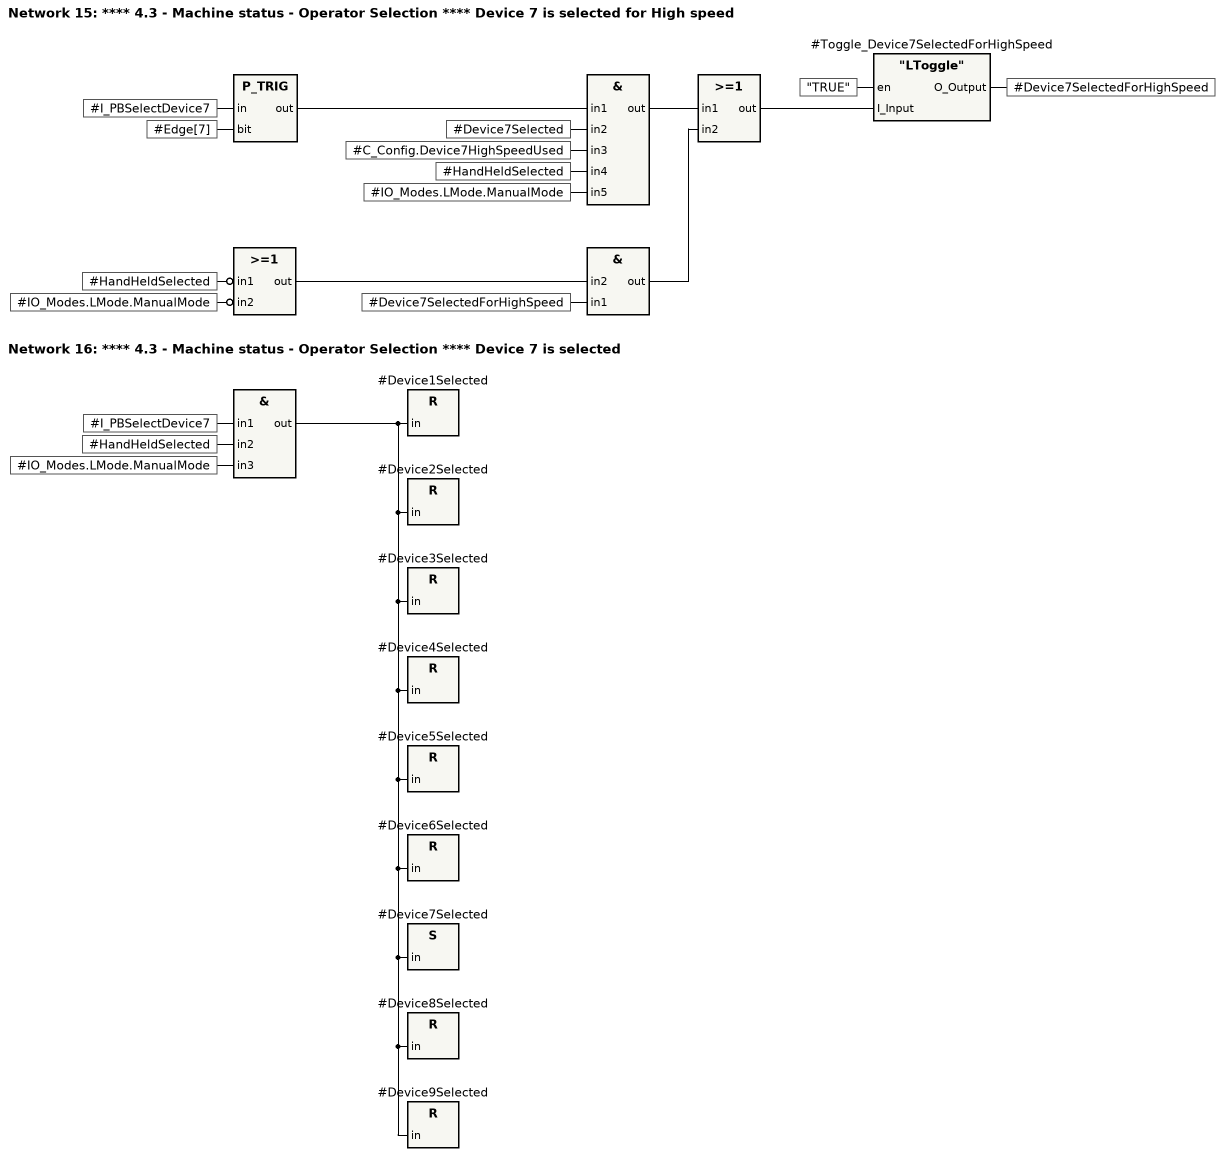
   #_w1 := #I_PBSelectDevice7 AND NOT #Edge[7];   // rising edge
   #Edge[7] := #I_PBSelectDevice7;
   IF "TRUE" THEN
       #Toggle_Device7SelectedForHighSpeed(I_Input := (#_w1 AND #Device7Selected AND #C_Config.Device7HighSpeedUsed AND #HandHeldSelected AND #IO_Modes.LMode.ManualMode) OR ((NOT #HandHeldSelected OR NOT #IO_Modes.LMode.ManualMode) AND #Device7SelectedForHighSpeed),   // "LToggle"
                               O_Output => #Device7SelectedForHighSpeed);
   END_IF;
END_REGION

REGION Network 16: **** 4.3 - Machine status - Operator Selection **** Device 7 is selected
   IF #I_PBSelectDevice7 AND #HandHeldSelected AND #IO_Modes.LMode.ManualMode THEN
       #Device1Selected := FALSE;
       #Device2Selected := FALSE;
       #Device3Selected := FALSE;
       #Device4Selected := FALSE;
       #Device5Selected := FALSE;
       #Device6Selected := FALSE;
       #Device7Selected := TRUE;
       #Device8Selected := FALSE;
       #Device9Selected := FALSE;
   END_IF;
END_REGION

REGION Network 17: **** 4.3 - Machine status - Operator Selection **** Device 8 is selected for High speed
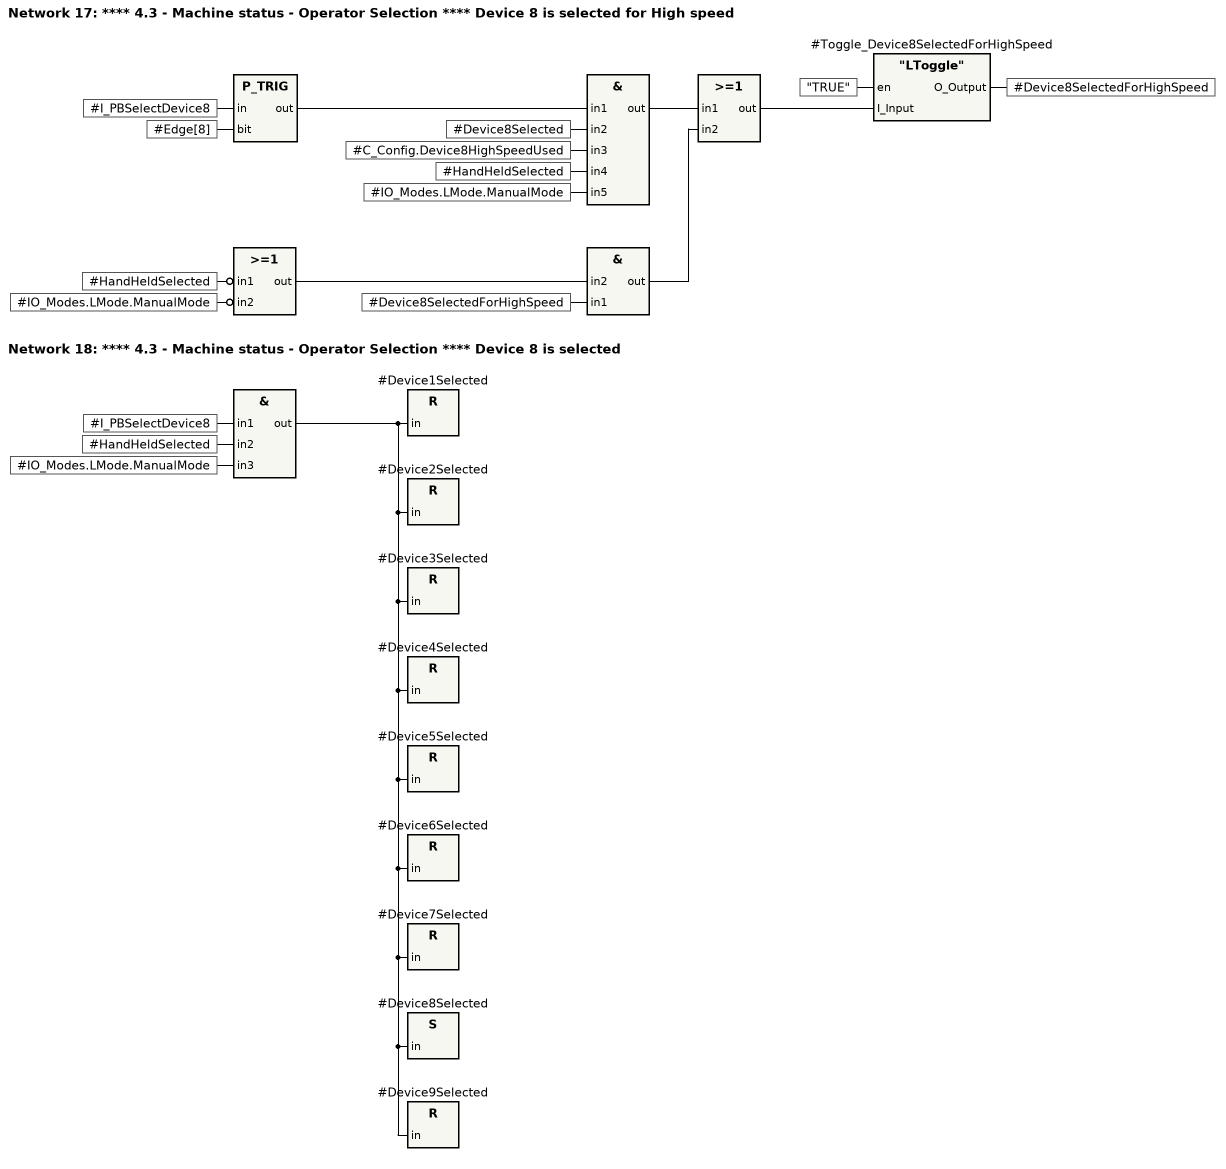
   #_w1 := #I_PBSelectDevice8 AND NOT #Edge[8];   // rising edge
   #Edge[8] := #I_PBSelectDevice8;
   IF "TRUE" THEN
       #Toggle_Device8SelectedForHighSpeed(I_Input := (#_w1 AND #Device8Selected AND #C_Config.Device8HighSpeedUsed AND #HandHeldSelected AND #IO_Modes.LMode.ManualMode) OR ((NOT #HandHeldSelected OR NOT #IO_Modes.LMode.ManualMode) AND #Device8SelectedForHighSpeed),   // "LToggle"
                               O_Output => #Device8SelectedForHighSpeed);
   END_IF;
END_REGION

REGION Network 18: **** 4.3 - Machine status - Operator Selection **** Device 8 is selected
   IF #I_PBSelectDevice8 AND #HandHeldSelected AND #IO_Modes.LMode.ManualMode THEN
       #Device1Selected := FALSE;
       #Device2Selected := FALSE;
       #Device3Selected := FALSE;
       #Device4Selected := FALSE;
       #Device5Selected := FALSE;
       #Device6Selected := FALSE;
       #Device7Selected := FALSE;
       #Device8Selected := TRUE;
       #Device9Selected := FALSE;
   END_IF;
END_REGION

REGION Network 19: **** 4.3 - Machine status - Operator Selection **** Device 9 is selected for High speed
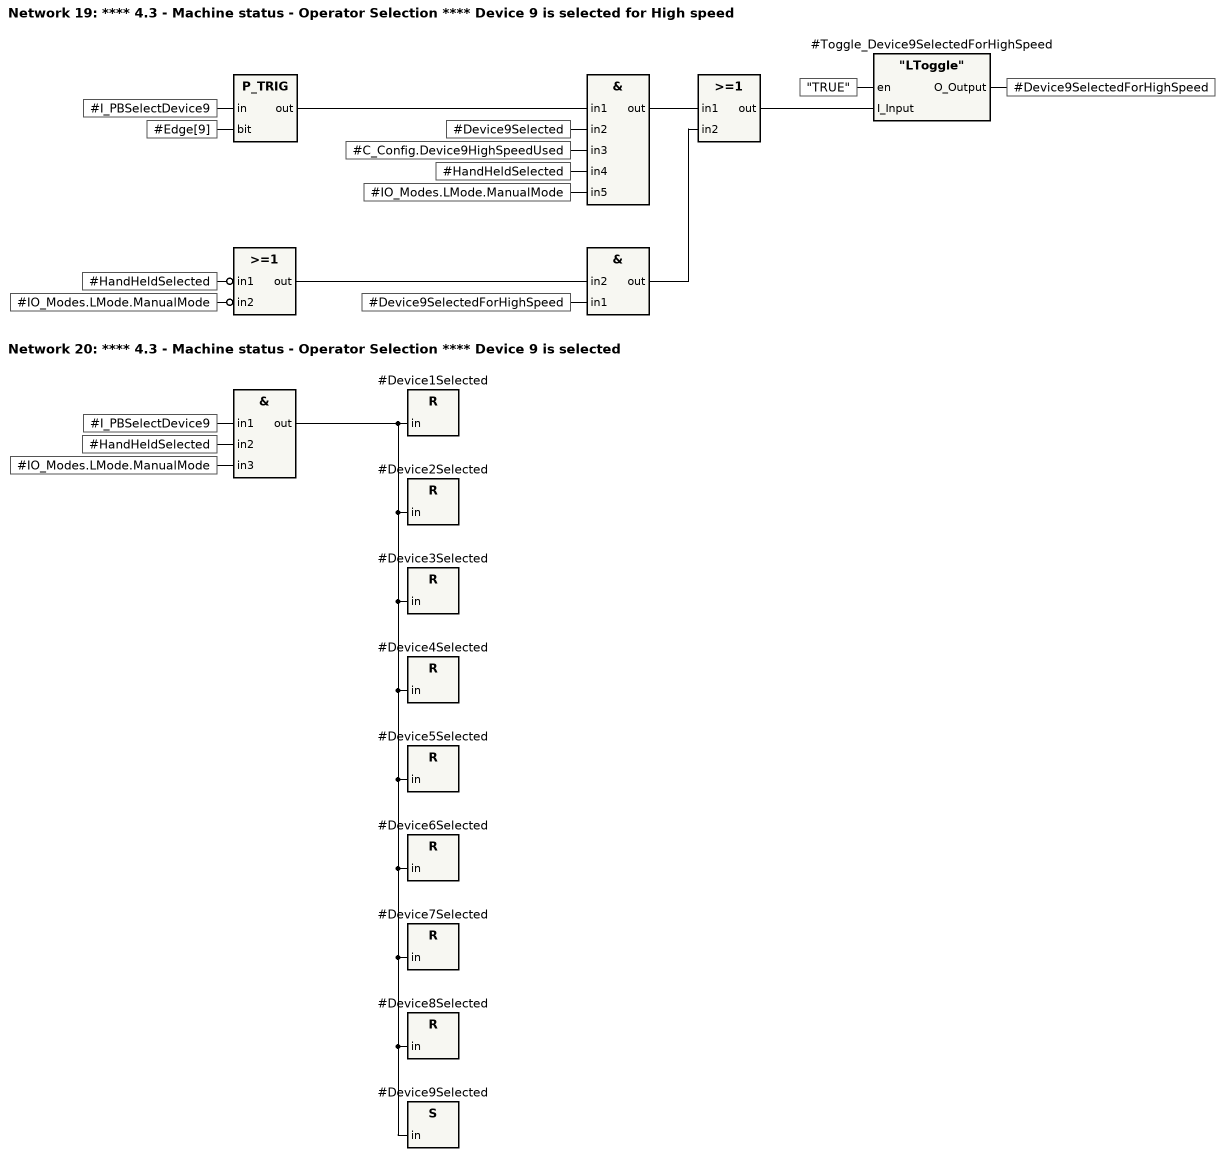
   #_w1 := #I_PBSelectDevice9 AND NOT #Edge[9];   // rising edge
   #Edge[9] := #I_PBSelectDevice9;
   IF "TRUE" THEN
       #Toggle_Device9SelectedForHighSpeed(I_Input := (#_w1 AND #Device9Selected AND #C_Config.Device9HighSpeedUsed AND #HandHeldSelected AND #IO_Modes.LMode.ManualMode) OR ((NOT #HandHeldSelected OR NOT #IO_Modes.LMode.ManualMode) AND #Device9SelectedForHighSpeed),   // "LToggle"
                               O_Output => #Device9SelectedForHighSpeed);
   END_IF;
END_REGION

REGION Network 20: **** 4.3 - Machine status - Operator Selection **** Device 9 is selected
   IF #I_PBSelectDevice9 AND #HandHeldSelected AND #IO_Modes.LMode.ManualMode THEN
       #Device1Selected := FALSE;
       #Device2Selected := FALSE;
       #Device3Selected := FALSE;
       #Device4Selected := FALSE;
       #Device5Selected := FALSE;
       #Device6Selected := FALSE;
       #Device7Selected := FALSE;
       #Device8Selected := FALSE;
       #Device9Selected := TRUE;
   END_IF;
END_REGION

REGION Network 21: **** 4.6 - Machine Status - Indication **** Indication Push button Device 1
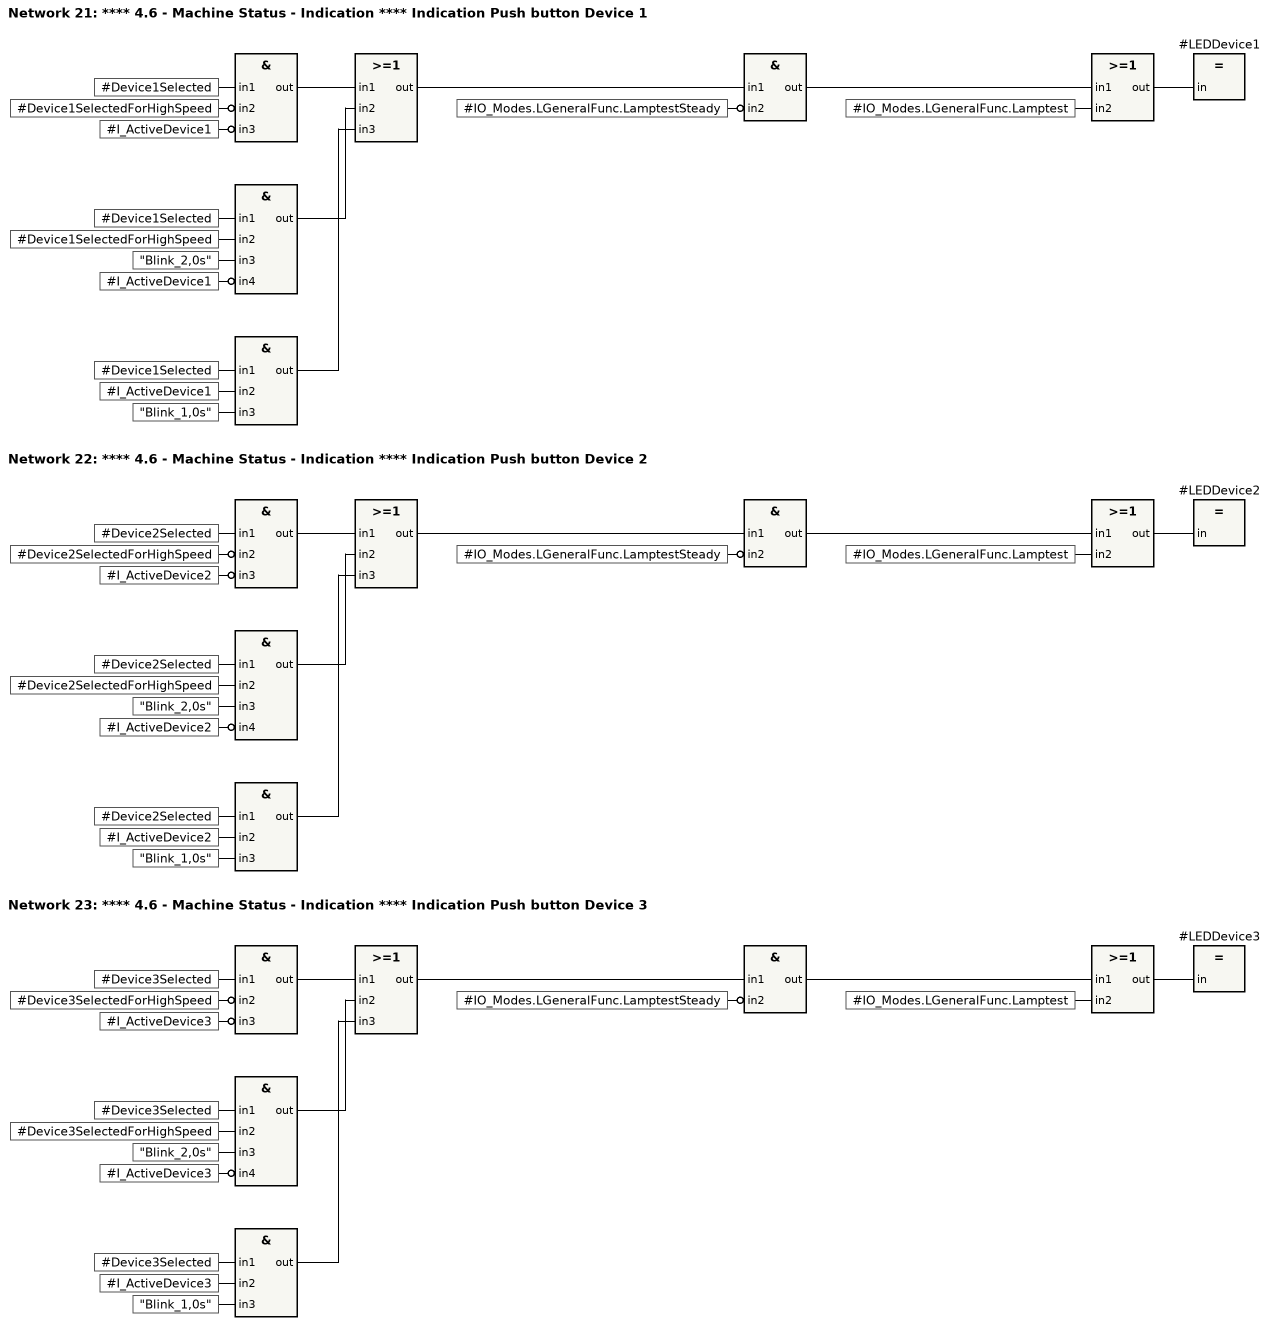
   #LEDDevice1 := (((#Device1Selected AND NOT #Device1SelectedForHighSpeed AND NOT #I_ActiveDevice1) OR (#Device1Selected AND #Device1SelectedForHighSpeed AND "Blink_2,0s" AND NOT #I_ActiveDevice1) OR (#Device1Selected AND #I_ActiveDevice1 AND "Blink_1,0s")) AND NOT #IO_Modes.LGeneralFunc.LamptestSteady) OR #IO_Modes.LGeneralFunc.Lamptest;
END_REGION

REGION Network 22: **** 4.6 - Machine Status - Indication **** Indication Push button Device 2
   #LEDDevice2 := (((#Device2Selected AND NOT #Device2SelectedForHighSpeed AND NOT #I_ActiveDevice2) OR (#Device2Selected AND #Device2SelectedForHighSpeed AND "Blink_2,0s" AND NOT #I_ActiveDevice2) OR (#Device2Selected AND #I_ActiveDevice2 AND "Blink_1,0s")) AND NOT #IO_Modes.LGeneralFunc.LamptestSteady) OR #IO_Modes.LGeneralFunc.Lamptest;
END_REGION

REGION Network 23: **** 4.6 - Machine Status - Indication **** Indication Push button Device 3
   #LEDDevice3 := (((#Device3Selected AND NOT #Device3SelectedForHighSpeed AND NOT #I_ActiveDevice3) OR (#Device3Selected AND #Device3SelectedForHighSpeed AND "Blink_2,0s" AND NOT #I_ActiveDevice3) OR (#Device3Selected AND #I_ActiveDevice3 AND "Blink_1,0s")) AND NOT #IO_Modes.LGeneralFunc.LamptestSteady) OR #IO_Modes.LGeneralFunc.Lamptest;
END_REGION

REGION Network 24: **** 4.6 - Machine Status - Indication **** Indication Push button Device 4
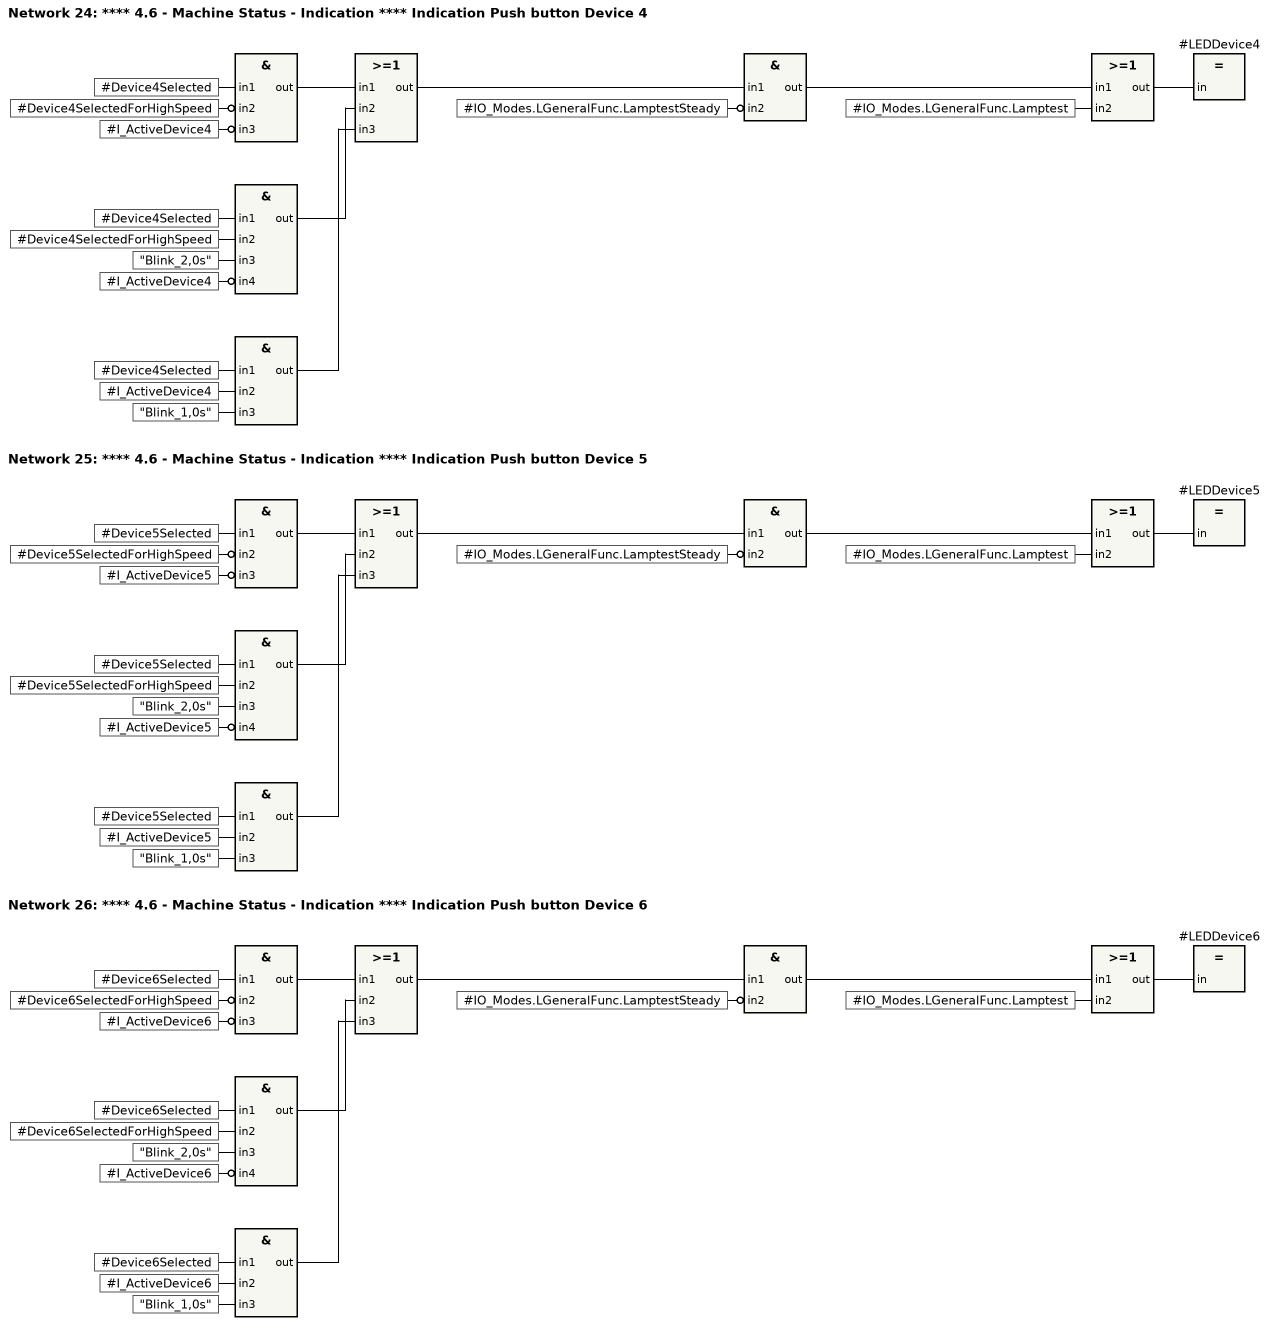
   #LEDDevice4 := (((#Device4Selected AND NOT #Device4SelectedForHighSpeed AND NOT #I_ActiveDevice4) OR (#Device4Selected AND #Device4SelectedForHighSpeed AND "Blink_2,0s" AND NOT #I_ActiveDevice4) OR (#Device4Selected AND #I_ActiveDevice4 AND "Blink_1,0s")) AND NOT #IO_Modes.LGeneralFunc.LamptestSteady) OR #IO_Modes.LGeneralFunc.Lamptest;
END_REGION

REGION Network 25: **** 4.6 - Machine Status - Indication **** Indication Push button Device 5
   #LEDDevice5 := (((#Device5Selected AND NOT #Device5SelectedForHighSpeed AND NOT #I_ActiveDevice5) OR (#Device5Selected AND #Device5SelectedForHighSpeed AND "Blink_2,0s" AND NOT #I_ActiveDevice5) OR (#Device5Selected AND #I_ActiveDevice5 AND "Blink_1,0s")) AND NOT #IO_Modes.LGeneralFunc.LamptestSteady) OR #IO_Modes.LGeneralFunc.Lamptest;
END_REGION

REGION Network 26: **** 4.6 - Machine Status - Indication **** Indication Push button Device 6
   #LEDDevice6 := (((#Device6Selected AND NOT #Device6SelectedForHighSpeed AND NOT #I_ActiveDevice6) OR (#Device6Selected AND #Device6SelectedForHighSpeed AND "Blink_2,0s" AND NOT #I_ActiveDevice6) OR (#Device6Selected AND #I_ActiveDevice6 AND "Blink_1,0s")) AND NOT #IO_Modes.LGeneralFunc.LamptestSteady) OR #IO_Modes.LGeneralFunc.Lamptest;
END_REGION

REGION Network 27: **** 4.6 - Machine Status - Indication **** Indication Push button Device 7
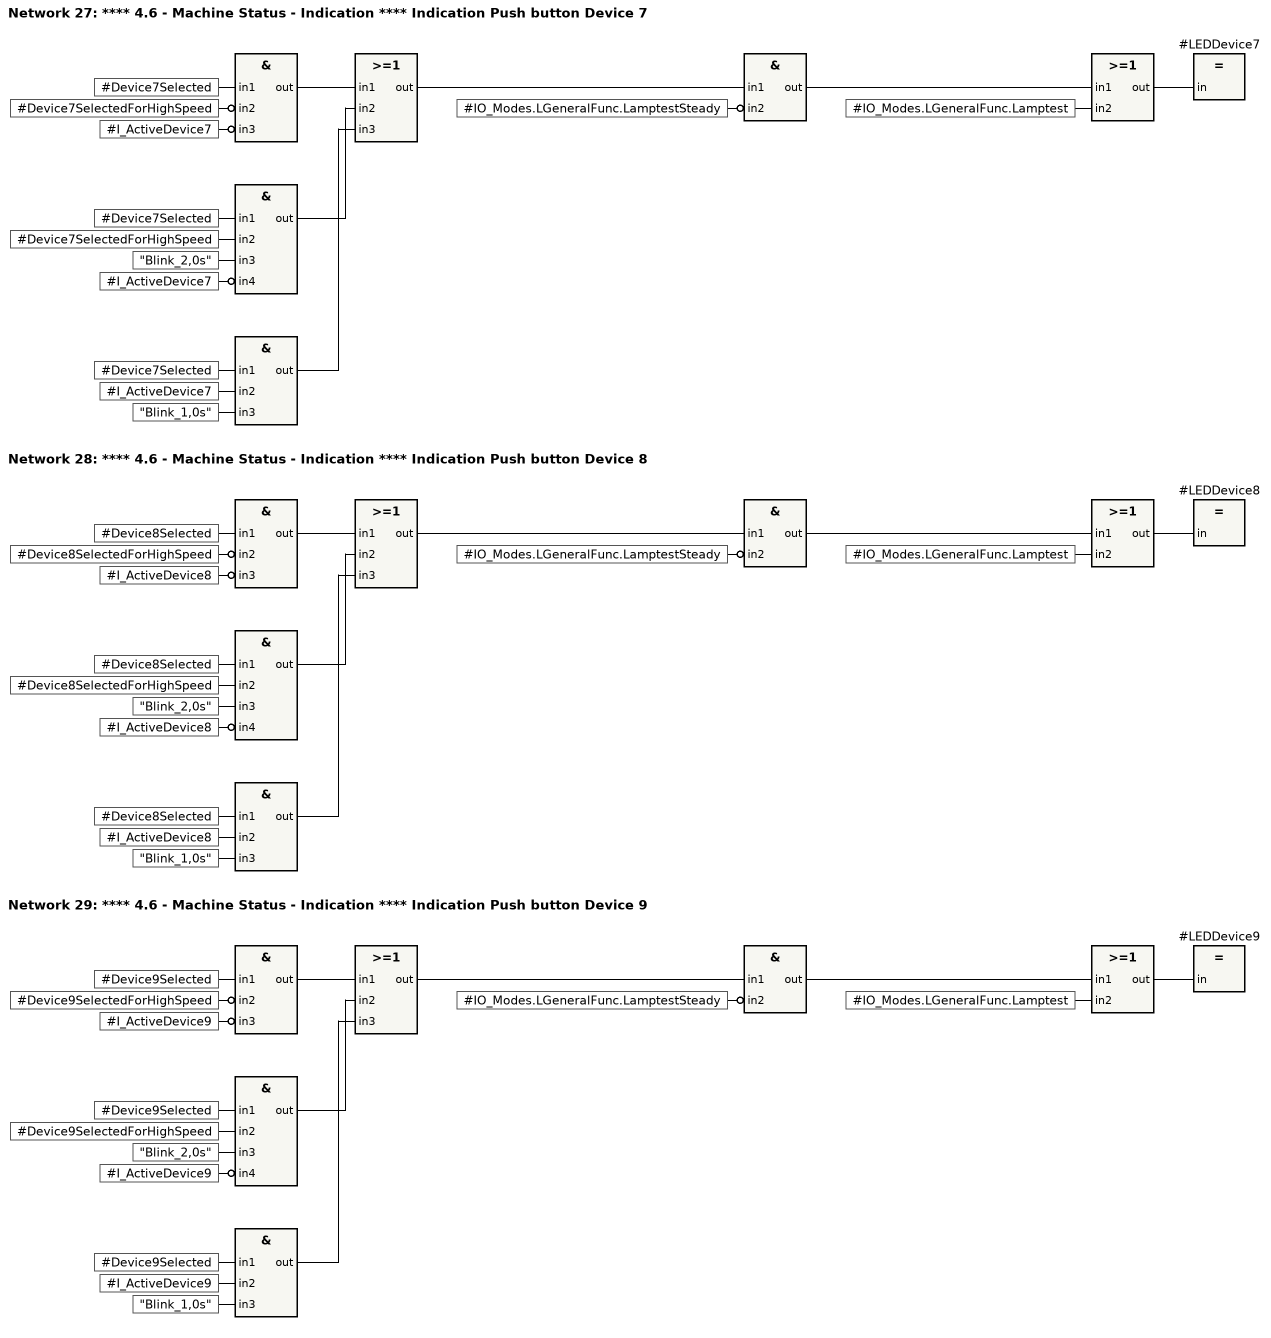
   #LEDDevice7 := (((#Device7Selected AND NOT #Device7SelectedForHighSpeed AND NOT #I_ActiveDevice7) OR (#Device7Selected AND #Device7SelectedForHighSpeed AND "Blink_2,0s" AND NOT #I_ActiveDevice7) OR (#Device7Selected AND #I_ActiveDevice7 AND "Blink_1,0s")) AND NOT #IO_Modes.LGeneralFunc.LamptestSteady) OR #IO_Modes.LGeneralFunc.Lamptest;
END_REGION

REGION Network 28: **** 4.6 - Machine Status - Indication **** Indication Push button Device 8
   #LEDDevice8 := (((#Device8Selected AND NOT #Device8SelectedForHighSpeed AND NOT #I_ActiveDevice8) OR (#Device8Selected AND #Device8SelectedForHighSpeed AND "Blink_2,0s" AND NOT #I_ActiveDevice8) OR (#Device8Selected AND #I_ActiveDevice8 AND "Blink_1,0s")) AND NOT #IO_Modes.LGeneralFunc.LamptestSteady) OR #IO_Modes.LGeneralFunc.Lamptest;
END_REGION

REGION Network 29: **** 4.6 - Machine Status - Indication **** Indication Push button Device 9
   #LEDDevice9 := (((#Device9Selected AND NOT #Device9SelectedForHighSpeed AND NOT #I_ActiveDevice9) OR (#Device9Selected AND #Device9SelectedForHighSpeed AND "Blink_2,0s" AND NOT #I_ActiveDevice9) OR (#Device9Selected AND #I_ActiveDevice9 AND "Blink_1,0s")) AND NOT #IO_Modes.LGeneralFunc.LamptestSteady) OR #IO_Modes.LGeneralFunc.Lamptest;
END_REGION

REGION Network 30: **** 5.2 - Equations **** High Speed Selected
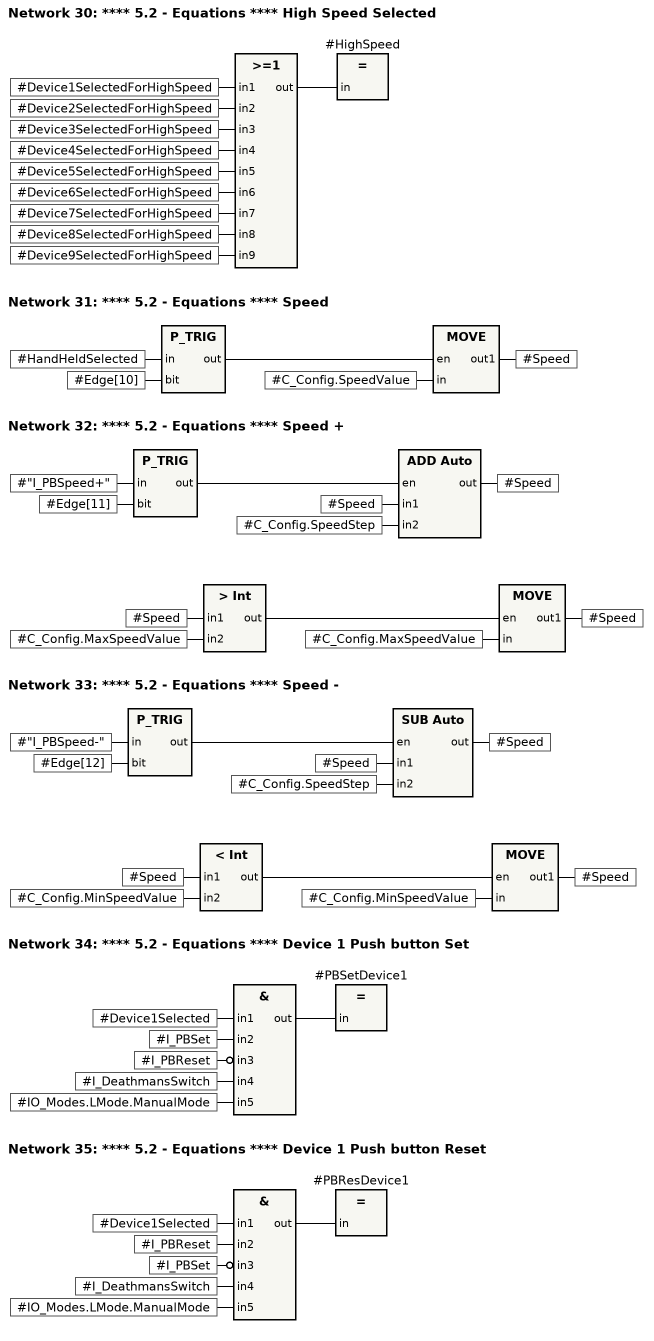
   #HighSpeed := #Device1SelectedForHighSpeed OR #Device2SelectedForHighSpeed OR #Device3SelectedForHighSpeed OR #Device4SelectedForHighSpeed OR #Device5SelectedForHighSpeed OR #Device6SelectedForHighSpeed OR #Device7SelectedForHighSpeed OR #Device8SelectedForHighSpeed OR #Device9SelectedForHighSpeed;
END_REGION

REGION Network 31: **** 5.2 - Equations **** Speed
   #_w1 := #HandHeldSelected AND NOT #Edge[10];   // rising edge
   #Edge[10] := #HandHeldSelected;
   IF #_w1 THEN #Speed := #C_Config.SpeedValue; END_IF;
END_REGION

REGION Network 32: **** 5.2 - Equations **** Speed +
   #_w1 := #"I_PBSpeed+" AND NOT #Edge[11];   // rising edge
   #Edge[11] := #"I_PBSpeed+";
   IF #_w1 THEN #Speed := #Speed + #C_Config.SpeedStep; END_IF;
   IF #Speed > #C_Config.MaxSpeedValue THEN #Speed := #C_Config.MaxSpeedValue; END_IF;
END_REGION

REGION Network 33: **** 5.2 - Equations **** Speed -
   #_w1 := #"I_PBSpeed-" AND NOT #Edge[12];   // rising edge
   #Edge[12] := #"I_PBSpeed-";
   IF #_w1 THEN #Speed := #Speed - #C_Config.SpeedStep; END_IF;
   IF #Speed < #C_Config.MinSpeedValue THEN #Speed := #C_Config.MinSpeedValue; END_IF;
END_REGION

REGION Network 34: **** 5.2 - Equations **** Device 1 Push button Set
   #PBSetDevice1 := #Device1Selected AND #I_PBSet AND NOT #I_PBReset AND #I_DeathmansSwitch AND #IO_Modes.LMode.ManualMode;
END_REGION

REGION Network 35: **** 5.2 - Equations **** Device 1 Push button Reset
   #PBResDevice1 := #Device1Selected AND #I_PBReset AND NOT #I_PBSet AND #I_DeathmansSwitch AND #IO_Modes.LMode.ManualMode;
END_REGION

REGION Network 36: **** 5.2 - Equations **** Device 2 Push button Set
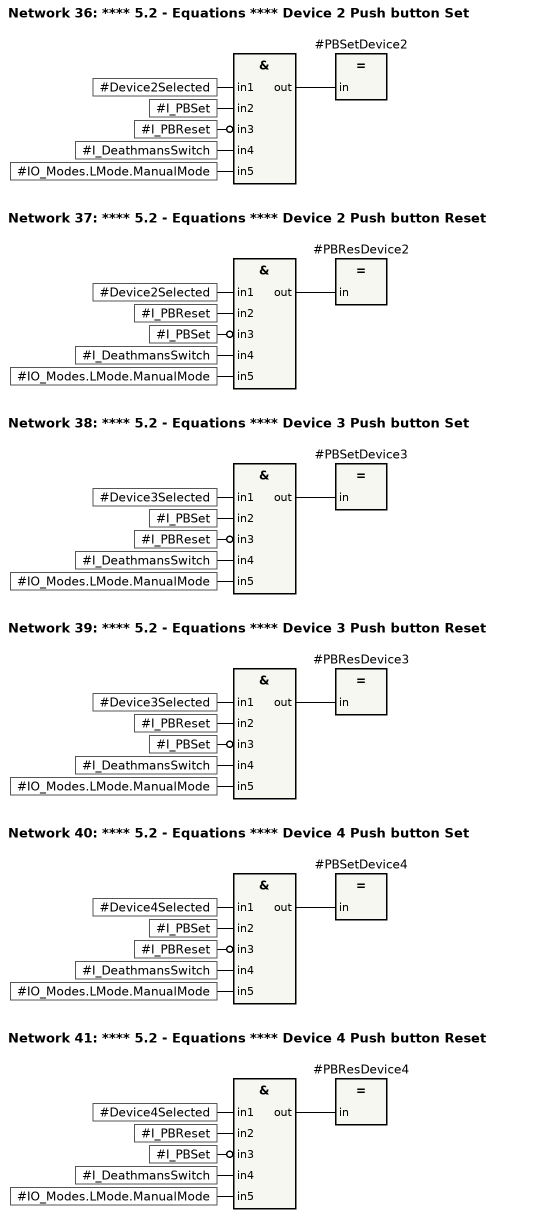
   #PBSetDevice2 := #Device2Selected AND #I_PBSet AND NOT #I_PBReset AND #I_DeathmansSwitch AND #IO_Modes.LMode.ManualMode;
END_REGION

REGION Network 37: **** 5.2 - Equations **** Device 2 Push button Reset
   #PBResDevice2 := #Device2Selected AND #I_PBReset AND NOT #I_PBSet AND #I_DeathmansSwitch AND #IO_Modes.LMode.ManualMode;
END_REGION

REGION Network 38: **** 5.2 - Equations **** Device 3 Push button Set
   #PBSetDevice3 := #Device3Selected AND #I_PBSet AND NOT #I_PBReset AND #I_DeathmansSwitch AND #IO_Modes.LMode.ManualMode;
END_REGION

REGION Network 39: **** 5.2 - Equations **** Device 3 Push button Reset
   #PBResDevice3 := #Device3Selected AND #I_PBReset AND NOT #I_PBSet AND #I_DeathmansSwitch AND #IO_Modes.LMode.ManualMode;
END_REGION

REGION Network 40: **** 5.2 - Equations **** Device 4 Push button Set
   #PBSetDevice4 := #Device4Selected AND #I_PBSet AND NOT #I_PBReset AND #I_DeathmansSwitch AND #IO_Modes.LMode.ManualMode;
END_REGION

REGION Network 41: **** 5.2 - Equations **** Device 4 Push button Reset
   #PBResDevice4 := #Device4Selected AND #I_PBReset AND NOT #I_PBSet AND #I_DeathmansSwitch AND #IO_Modes.LMode.ManualMode;
END_REGION

REGION Network 42: **** 5.2 - Equations **** Device 5 Push button Set
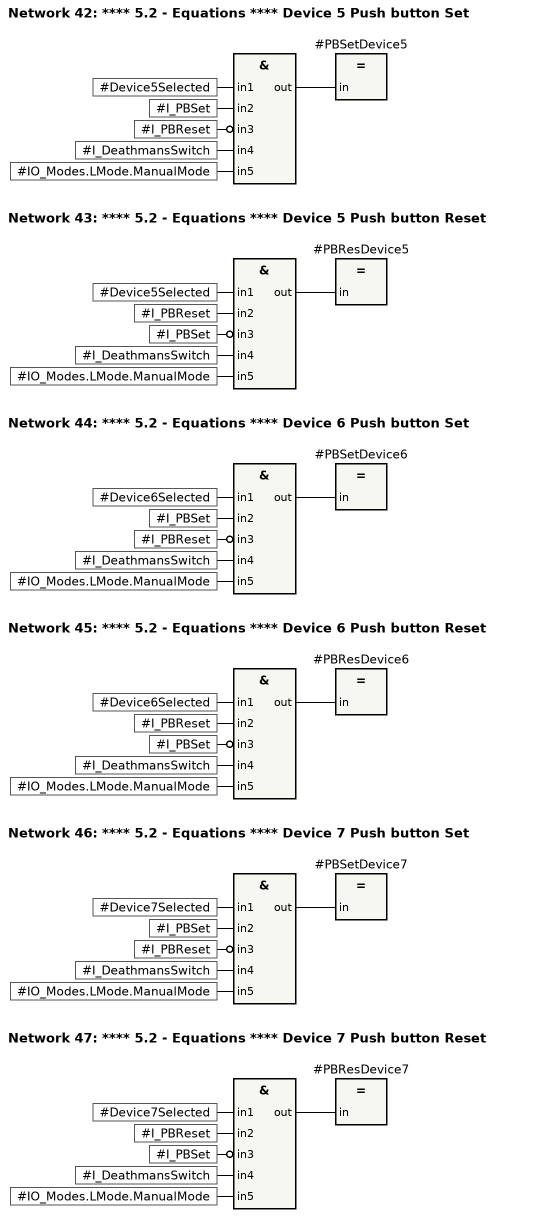
   #PBSetDevice5 := #Device5Selected AND #I_PBSet AND NOT #I_PBReset AND #I_DeathmansSwitch AND #IO_Modes.LMode.ManualMode;
END_REGION

REGION Network 43: **** 5.2 - Equations **** Device 5 Push button Reset
   #PBResDevice5 := #Device5Selected AND #I_PBReset AND NOT #I_PBSet AND #I_DeathmansSwitch AND #IO_Modes.LMode.ManualMode;
END_REGION

REGION Network 44: **** 5.2 - Equations **** Device 6 Push button Set
   #PBSetDevice6 := #Device6Selected AND #I_PBSet AND NOT #I_PBReset AND #I_DeathmansSwitch AND #IO_Modes.LMode.ManualMode;
END_REGION

REGION Network 45: **** 5.2 - Equations **** Device 6 Push button Reset
   #PBResDevice6 := #Device6Selected AND #I_PBReset AND NOT #I_PBSet AND #I_DeathmansSwitch AND #IO_Modes.LMode.ManualMode;
END_REGION

REGION Network 46: **** 5.2 - Equations **** Device 7 Push button Set
   #PBSetDevice7 := #Device7Selected AND #I_PBSet AND NOT #I_PBReset AND #I_DeathmansSwitch AND #IO_Modes.LMode.ManualMode;
END_REGION

REGION Network 47: **** 5.2 - Equations **** Device 7 Push button Reset
   #PBResDevice7 := #Device7Selected AND #I_PBReset AND NOT #I_PBSet AND #I_DeathmansSwitch AND #IO_Modes.LMode.ManualMode;
END_REGION

REGION Network 48: **** 5.2 - Equations **** Device 8 Push button Set
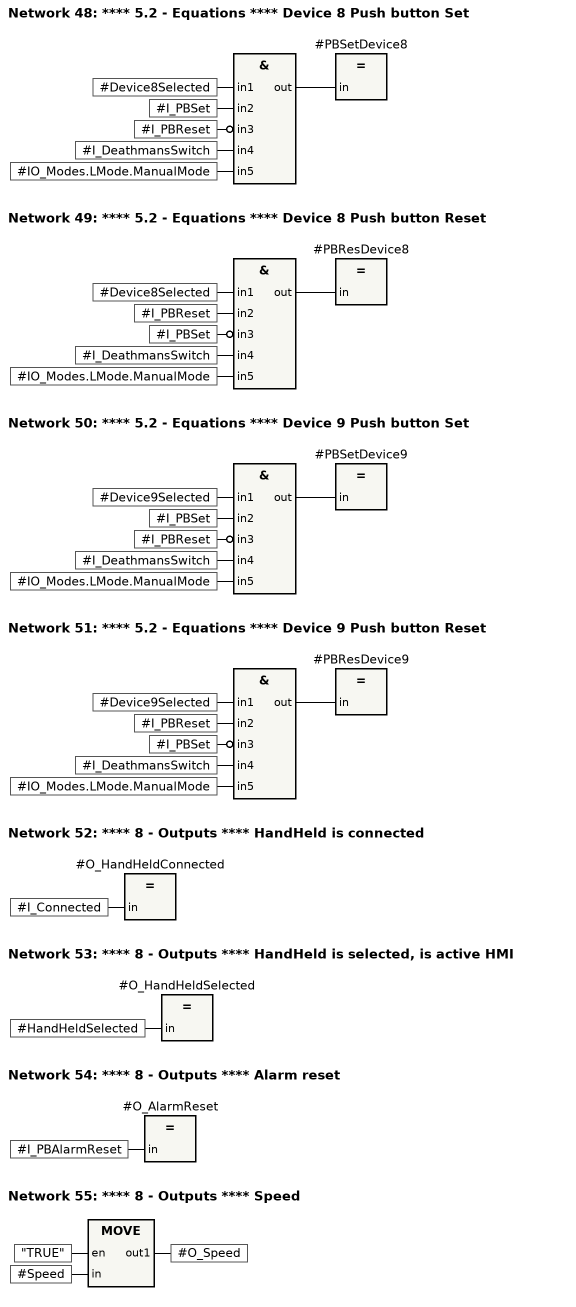
   #PBSetDevice8 := #Device8Selected AND #I_PBSet AND NOT #I_PBReset AND #I_DeathmansSwitch AND #IO_Modes.LMode.ManualMode;
END_REGION

REGION Network 49: **** 5.2 - Equations **** Device 8 Push button Reset
   #PBResDevice8 := #Device8Selected AND #I_PBReset AND NOT #I_PBSet AND #I_DeathmansSwitch AND #IO_Modes.LMode.ManualMode;
END_REGION

REGION Network 50: **** 5.2 - Equations **** Device 9 Push button Set
   #PBSetDevice9 := #Device9Selected AND #I_PBSet AND NOT #I_PBReset AND #I_DeathmansSwitch AND #IO_Modes.LMode.ManualMode;
END_REGION

REGION Network 51: **** 5.2 - Equations **** Device 9 Push button Reset
   #PBResDevice9 := #Device9Selected AND #I_PBReset AND NOT #I_PBSet AND #I_DeathmansSwitch AND #IO_Modes.LMode.ManualMode;
END_REGION

REGION Network 52: **** 8 - Outputs **** HandHeld is connected
   #O_HandHeldConnected := #I_Connected;
END_REGION

REGION Network 53: **** 8 - Outputs **** HandHeld is selected, is active HMI
   #O_HandHeldSelected := #HandHeldSelected;
END_REGION

REGION Network 54: **** 8 - Outputs **** Alarm reset
   #O_AlarmReset := #I_PBAlarmReset;
END_REGION

REGION Network 55: **** 8 - Outputs **** Speed
   IF "TRUE" THEN #O_Speed := #Speed; END_IF;
END_REGION

REGION Network 56: **** 8 - Outputs **** Speed+
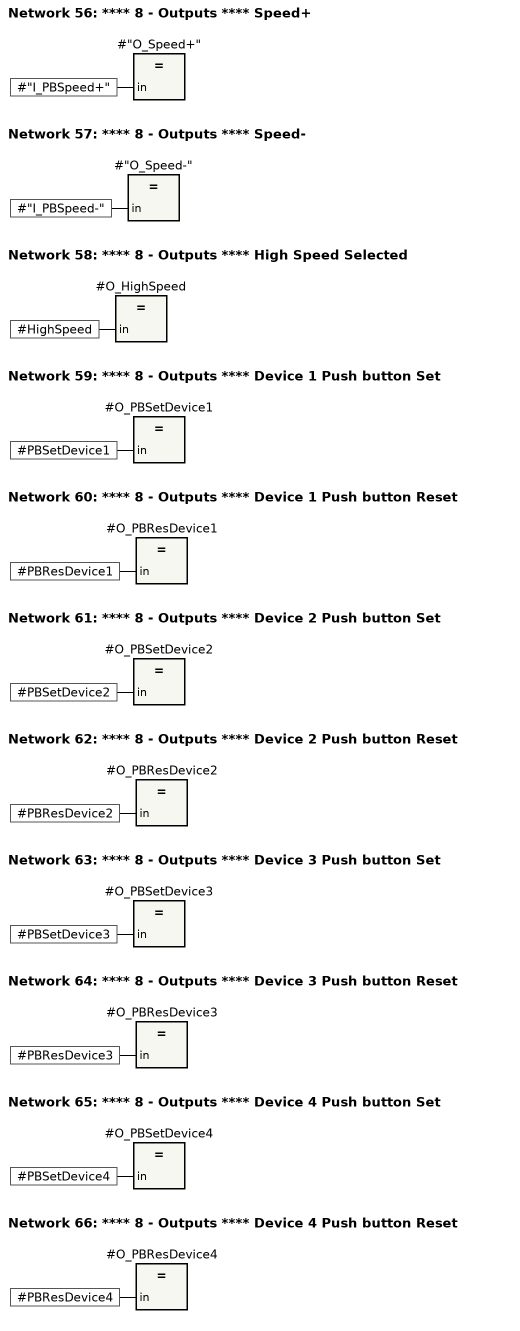
   #"O_Speed+" := #"I_PBSpeed+";
END_REGION

REGION Network 57: **** 8 - Outputs **** Speed-
   #"O_Speed-" := #"I_PBSpeed-";
END_REGION

REGION Network 58: **** 8 - Outputs **** High Speed Selected
   #O_HighSpeed := #HighSpeed;
END_REGION

REGION Network 59: **** 8 - Outputs **** Device 1 Push button Set
   #O_PBSetDevice1 := #PBSetDevice1;
END_REGION

REGION Network 60: **** 8 - Outputs **** Device 1 Push button Reset
   #O_PBResDevice1 := #PBResDevice1;
END_REGION

REGION Network 61: **** 8 - Outputs **** Device 2 Push button Set
   #O_PBSetDevice2 := #PBSetDevice2;
END_REGION

REGION Network 62: **** 8 - Outputs **** Device 2 Push button Reset
   #O_PBResDevice2 := #PBResDevice2;
END_REGION

REGION Network 63: **** 8 - Outputs **** Device 3 Push button Set
   #O_PBSetDevice3 := #PBSetDevice3;
END_REGION

REGION Network 64: **** 8 - Outputs **** Device 3 Push button Reset
   #O_PBResDevice3 := #PBResDevice3;
END_REGION

REGION Network 65: **** 8 - Outputs **** Device 4 Push button Set
   #O_PBSetDevice4 := #PBSetDevice4;
END_REGION

REGION Network 66: **** 8 - Outputs **** Device 4 Push button Reset
   #O_PBResDevice4 := #PBResDevice4;
END_REGION

REGION Network 67: **** 8 - Outputs **** Device 5 Push button Set
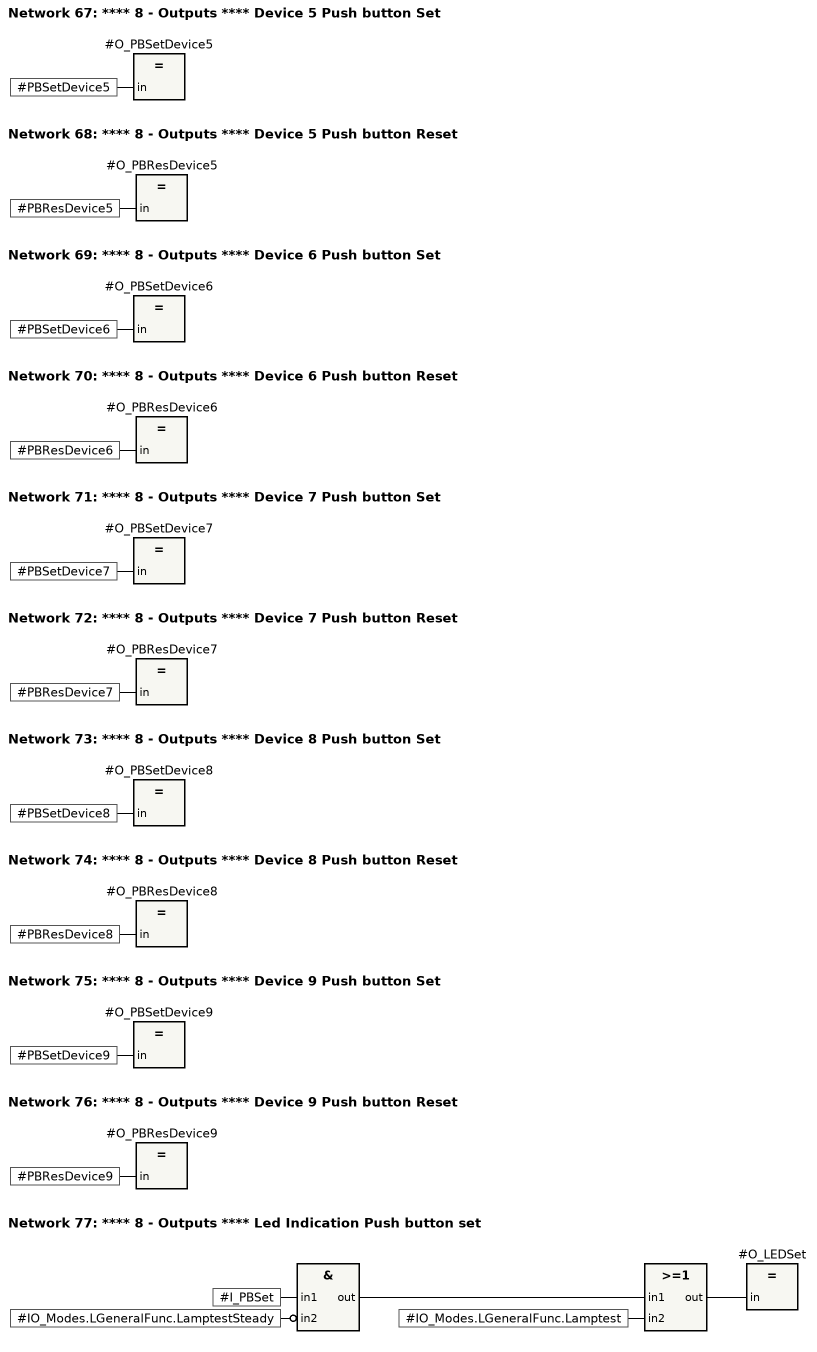
   #O_PBSetDevice5 := #PBSetDevice5;
END_REGION

REGION Network 68: **** 8 - Outputs **** Device 5 Push button Reset
   #O_PBResDevice5 := #PBResDevice5;
END_REGION

REGION Network 69: **** 8 - Outputs **** Device 6 Push button Set
   #O_PBSetDevice6 := #PBSetDevice6;
END_REGION

REGION Network 70: **** 8 - Outputs **** Device 6 Push button Reset
   #O_PBResDevice6 := #PBResDevice6;
END_REGION

REGION Network 71: **** 8 - Outputs **** Device 7 Push button Set
   #O_PBSetDevice7 := #PBSetDevice7;
END_REGION

REGION Network 72: **** 8 - Outputs **** Device 7 Push button Reset
   #O_PBResDevice7 := #PBResDevice7;
END_REGION

REGION Network 73: **** 8 - Outputs **** Device 8 Push button Set
   #O_PBSetDevice8 := #PBSetDevice8;
END_REGION

REGION Network 74: **** 8 - Outputs **** Device 8 Push button Reset
   #O_PBResDevice8 := #PBResDevice8;
END_REGION

REGION Network 75: **** 8 - Outputs **** Device 9 Push button Set
   #O_PBSetDevice9 := #PBSetDevice9;
END_REGION

REGION Network 76: **** 8 - Outputs **** Device 9 Push button Reset
   #O_PBResDevice9 := #PBResDevice9;
END_REGION

REGION Network 77: **** 8 - Outputs **** Led Indication Push button set
   #O_LEDSet := (#I_PBSet AND NOT #IO_Modes.LGeneralFunc.LamptestSteady) OR #IO_Modes.LGeneralFunc.Lamptest;
END_REGION

REGION Network 78: **** 8 - Outputs **** Led Indication Push button reset
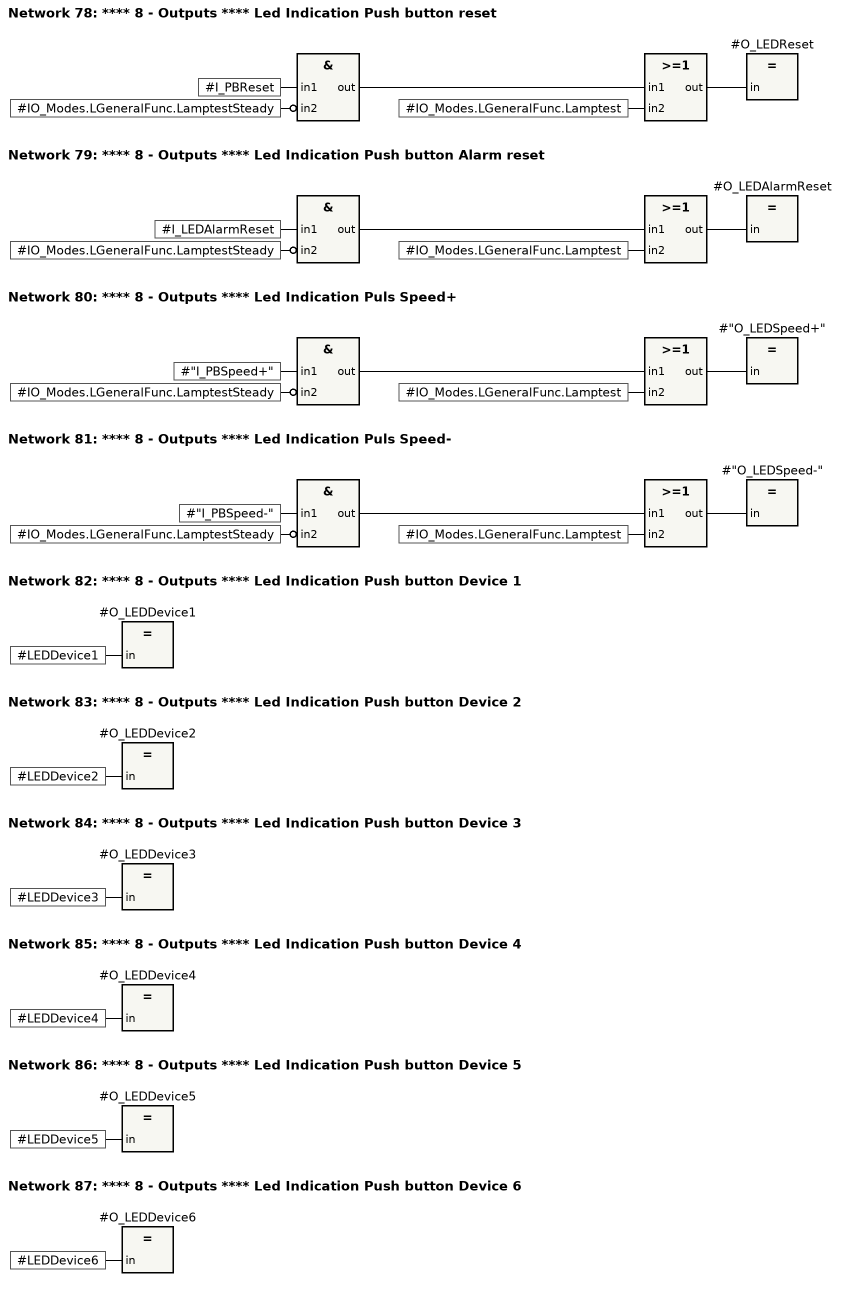
   #O_LEDReset := (#I_PBReset AND NOT #IO_Modes.LGeneralFunc.LamptestSteady) OR #IO_Modes.LGeneralFunc.Lamptest;
END_REGION

REGION Network 79: **** 8 - Outputs **** Led Indication Push button Alarm reset
   #O_LEDAlarmReset := (#I_LEDAlarmReset AND NOT #IO_Modes.LGeneralFunc.LamptestSteady) OR #IO_Modes.LGeneralFunc.Lamptest;
END_REGION

REGION Network 80: **** 8 - Outputs **** Led Indication Puls Speed+
   #"O_LEDSpeed+" := (#"I_PBSpeed+" AND NOT #IO_Modes.LGeneralFunc.LamptestSteady) OR #IO_Modes.LGeneralFunc.Lamptest;
END_REGION

REGION Network 81: **** 8 - Outputs **** Led Indication Puls Speed-
   #"O_LEDSpeed-" := (#"I_PBSpeed-" AND NOT #IO_Modes.LGeneralFunc.LamptestSteady) OR #IO_Modes.LGeneralFunc.Lamptest;
END_REGION

REGION Network 82: **** 8 - Outputs **** Led Indication Push button Device 1
   #O_LEDDevice1 := #LEDDevice1;
END_REGION

REGION Network 83: **** 8 - Outputs **** Led Indication Push button Device 2
   #O_LEDDevice2 := #LEDDevice2;
END_REGION

REGION Network 84: **** 8 - Outputs **** Led Indication Push button Device 3
   #O_LEDDevice3 := #LEDDevice3;
END_REGION

REGION Network 85: **** 8 - Outputs **** Led Indication Push button Device 4
   #O_LEDDevice4 := #LEDDevice4;
END_REGION

REGION Network 86: **** 8 - Outputs **** Led Indication Push button Device 5
   #O_LEDDevice5 := #LEDDevice5;
END_REGION

REGION Network 87: **** 8 - Outputs **** Led Indication Push button Device 6
   #O_LEDDevice6 := #LEDDevice6;
END_REGION

REGION Network 88: **** 8 - Outputs **** Led Indication Push button Device 7
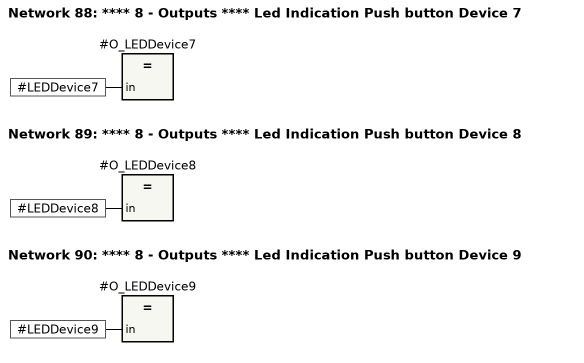
   #O_LEDDevice7 := #LEDDevice7;
END_REGION

REGION Network 89: **** 8 - Outputs **** Led Indication Push button Device 8
   #O_LEDDevice8 := #LEDDevice8;
END_REGION

REGION Network 90: **** 8 - Outputs **** Led Indication Push button Device 9
   #O_LEDDevice9 := #LEDDevice9;
END_REGION
END_FUNCTION_BLOCK
